LIN {X 0,Y 152.745,Z 601.305,A -85,B 0,C 180,E1 -23923.975,E2 -23923.975} C_VEL
LIN {X 0,Y 150.02,Z 597.18,A -85,B 0,C 180,E1 -23929.2,E2 -23929.2} C_VEL
LIN {X 0,Y 148.785,Z 591.816,A -85,B 0,C 180,E1 -23934.579,E2 -23934.579} C_VEL
LIN {X 0,Y 148.504,Z 586.8,A -85,B 0,C 180,E1 -23938.644,E2 -23938.644} C_VEL
LIN {X 0,Y 148.54,Z 579.677,A -85,B 0,C 180,E1 -23943.382,E2 -23943.382} C_VEL
LIN {X 0,Y 149.004,Z 570.731,A -85,B 0,C 180,E1 -23948.135,E2 -23948.135} C_VEL
LIN {X 0,Y 149.902,Z 561.531,A -85,B 0,C 180,E1 -23952.18,E2 -23952.18} C_VEL
LIN {X 0,Y 151.343,Z 550.54,A -85,B 0,C 180,E1 -23956.178,E2 -23956.178} C_VEL
LIN {X 0,Y 153.19,Z 538.222,A -85,B 0,C 180,E1 -23959.776,E2 -23959.776} C_VEL
LIN {X 0,Y 154.501,Z 528.967,A -85,B 0,C 180,E1 -23962.027,E2 -23962.027} C_VEL
LIN {X 0,Y 154.015,Z 524.912,A -85,B 0,C 180,E1 -23962.923,E2 -23962.923} C_VEL
LIN {X 0,Y 154.282,Z 525.794,A -85,B 0,C 180,E1 -23963.446,E2 -23963.446} C_VEL
LIN {X 0,Y 154.921,Z 526.142,A -85,B 0,C 180,E1 -23964.098,E2 -23964.098} C_VEL
LIN {X 0,Y 156.698,Z 525.145,A -85,B 0,C 180,E1 -23965.219,E2 -23965.219} C_VEL
LIN {X 0,Y 158.967,Z 522.474,A -85,B 0,C 180,E1 -23966.239,E2 -23966.239} C_VEL
LIN {X 0,Y 160.918,Z 521.843,A -85,B 0,C 180,E1 -23967.472,E2 -23967.472} C_VEL
LIN {X 0,Y 163.299,Z 519.845,A -85,B 0,C 180,E1 -23968.607,E2 -23968.607} C_VEL
LIN {X 0,Y 165.925,Z 516.496,A -85,B 0,C 180,E1 -23969.586,E2 -23969.586} C_VEL
LIN {X 0,Y 166.624,Z 515.781,A -85,B 0,C 180,E1 -23969.884,E2 -23969.884} C_VEL
LIN {X 0,Y 167.613,Z 515.285,A -85,B 0,C 180,E1 -23970.383,E2 -23970.383} C_VEL
LIN {X 0,Y 170.37,Z 518.349,A -85,B 0,C 180,E1 -23972.43,E2 -23972.43} C_VEL
LIN {X 0,Y 172.937,Z 522.605,A -85,B 0,C 180,E1 -23974.5,E2 -23974.5} C_VEL
LIN {X 0,Y 176.225,Z 530.359,A -85,B 0,C 180,E1 -23977.459,E2 -23977.459} C_VEL
LIN {X 0,Y 178.356,Z 536.742,A -85,B 0,C 180,E1 -23979.65,E2 -23979.65} C_VEL
LIN {X 0,Y 179.284,Z 542.682,A -85,B 0,C 180,E1 -23981.331,E2 -23981.331} C_VEL
LIN {X 0,Y 179.755,Z 554.232,A -85,B 0,C 180,E1 -23984.405,E2 -23984.405} C_VEL
LIN {X 0,Y 179.119,Z 565.311,A -85,B 0,C 180,E1 -23987.445,E2 -23987.445} C_VEL
LIN {X 0,Y 178.567,Z 569.644,A -85,B 0,C 180,E1 -23988.697,E2 -23988.697} C_VEL
LIN {X 0,Y 173.803,Z 580.088,A -85,B 0,C 180,E1 -23991.185,E2 -23991.185} C_VEL
LIN {X 0,Y 168.532,Z 590.306,A -85,B 0,C 180,E1 -23994.277,E2 -23994.277} C_VEL
LIN {X 0,Y 163.924,Z 598.73,A -85,B 0,C 180,E1 -23997.59,E2 -23997.59} C_VEL
LIN {X 0,Y 159.001,Z 606.865,A -85,B 0,C 180,E1 -24001.699,E2 -24001.699} C_VEL
LIN {X 0,Y 155.248,Z 613.225,A -85,B 0,C 180,E1 -24005.953,E2 -24005.953} C_VEL
LIN {X 0,Y 152.55,Z 617.694,A -85,B 0,C 180,E1 -24009.783,E2 -24009.783} C_VEL
LIN {X 0,Y 150.41,Z 621.2,A -85,B 0,C 180,E1 -24013.715,E2 -24013.715} C_VEL
LIN {X 0,Y 148.596,Z 624.62,A -85,B 0,C 180,E1 -24019.091,E2 -24019.091} C_VEL
LIN {X 0,Y 147.704,Z 626.652,A -85,B 0,C 180,E1 -24024.536,E2 -24024.536} C_VEL
LIN {X 0,Y 147.629,Z 627.344,A -85,B 0,C 180,E1 -24029.997,E2 -24029.997} C_VEL
LIN {X 0,Y 147.702,Z 626.705,A -85,B 0,C 180,E1 -24035.457,E2 -24035.457} C_VEL
LIN {X 0,Y 148.571,Z 624.718,A -85,B 0,C 180,E1 -24040.903,E2 -24040.903} C_VEL
LIN {X 0,Y 150.349,Z 621.341,A -85,B 0,C 180,E1 -24046.284,E2 -24046.284} C_VEL
LIN {X 0,Y 153.36,Z 616.469,A -85,B 0,C 180,E1 -24051.503,E2 -24051.503} C_VEL
LIN {X 0,Y 156.231,Z 611.748,A -85,B 0,C 180,E1 -24055.296,E2 -24055.296} C_VEL
LIN {X 0,Y 160.294,Z 604.906,A -85,B 0,C 180,E1 -24059.551,E2 -24059.551} C_VEL
LIN {X 0,Y 165.31,Z 596.406,A -85,B 0,C 180,E1 -24063.547,E2 -24063.547} C_VEL
LIN {X 0,Y 170.162,Z 587.512,A -85,B 0,C 180,E1 -24066.785,E2 -24066.785} C_VEL
LIN {X 0,Y 175.567,Z 576.736,A -85,B 0,C 180,E1 -24069.824,E2 -24069.824} C_VEL
LIN {X 0,Y 178.508,Z 570.135,A -85,B 0,C 180,E1 -24071.344,E2 -24071.344} C_VEL
LIN {X 0,Y 179.601,Z 561.031,A -85,B 0,C 180,E1 -24073.901,E2 -24073.901} C_VEL
LIN {X 0,Y 179.815,Z 552.025,A -85,B 0,C 180,E1 -24076.347,E2 -24076.347} C_VEL
LIN {X 0,Y 179.189,Z 541.022,A -85,B 0,C 180,E1 -24079.277,E2 -24079.277} C_VEL
LIN {X 0,Y 178.169,Z 535.607,A -85,B 0,C 180,E1 -24080.866,E2 -24080.866} C_VEL
LIN {X 0,Y 174.614,Z 526.074,A -85,B 0,C 180,E1 -24084.295,E2 -24084.295} C_VEL
LIN {X 0,Y 171.422,Z 519.258,A -85,B 0,C 180,E1 -24087.096,E2 -24087.096} C_VEL
LIN {X 0,Y 169.471,Z 515.528,A -85,B 0,C 180,E1 -24088.776,E2 -24088.776} C_VEL
LIN {X 0,Y 166.715,Z 510.789,A -85,B 0,C 180,E1 -24091.188,E2 -24091.188} C_VEL
LIN {X 0,Y 164.013,Z 506.647,A -85,B 0,C 180,E1 -24093.604,E2 -24093.604} C_VEL
LIN {X 0,Y 163.126,Z 505.162,A -85,B 0,C 180,E1 -24094.479,E2 -24094.479} C_VEL
LIN {X 0,Y 160.311,Z 501.441,A -85,B 0,C 180,E1 -24097.21,E2 -24097.21} C_VEL
LIN {X 0,Y 159.174,Z 499.399,A -85,B 0,C 180,E1 -24098.511,E2 -24098.511} C_VEL
LIN {X 0,Y 155.732,Z 495.52,A -85,B 0,C 180,E1 -24102.603,E2 -24102.603} C_VEL
LIN {X 0,Y 154.403,Z 493.061,A -85,B 0,C 180,E1 -24104.827,E2 -24104.827} C_VEL
LIN {X 0,Y 154.236,Z 491.472,A -85,B 0,C 180,E1 -24109.498,E2 -24109.498} C_VEL
LIN {X 0,Y 154.177,Z 490.844,A -85,B 0,C 180,E1 -24112.14,E2 -24112.14} C_VEL
LIN {X 0,Y 154.299,Z 489.663,A -85,B 0,C 180,E1 -24120,E2 -24120} C_VEL
LIN {X 0,Y 154.024,Z 490.167,A -85,B 0,C 180,E1 -24125.236,E2 -24125.236} C_VEL
LIN {X 0,Y 154.391,Z 491.072,A -85,B 0,C 180,E1 -24130.491,E2 -24130.491} C_VEL
LIN {X 0,Y 154.81,Z 492.811,A -85,B 0,C 180,E1 -24135.806,E2 -24135.806} C_VEL
LIN {X 0,Y 158.463,Z 497.876,A -85,B 0,C 180,E1 -24140.781,E2 -24140.781} C_VEL
LIN {X 0,Y 160.423,Z 499.793,A -85,B 0,C 180,E1 -24142.795,E2 -24142.795} C_VEL
LIN {X 0,Y 163.521,Z 504.046,A -85,B 0,C 180,E1 -24145.796,E2 -24145.796} C_VEL
LIN {X 0,Y 165.119,Z 505.889,A -85,B 0,C 180,E1 -24147.144,E2 -24147.144} C_VEL
LIN {X 0,Y 168.025,Z 510.29,A -85,B 0,C 180,E1 -24149.63,E2 -24149.63} C_VEL
LIN {X 0,Y 172.528,Z 517.457,A -85,B 0,C 180,E1 -24153.187,E2 -24153.187} C_VEL
LIN {X 0,Y 175.298,Z 522.617,A -85,B 0,C 180,E1 -24155.368,E2 -24155.368} C_VEL
LIN {X 0,Y 178.224,Z 530.027,A -85,B 0,C 180,E1 -24157.944,E2 -24157.944} C_VEL
LIN {X 0,Y 181.369,Z 540.405,A -85,B 0,C 180,E1 -24161.204,E2 -24161.204} C_VEL
LIN {X 0,Y 182.33,Z 544.543,A -85,B 0,C 180,E1 -24162.42,E2 -24162.42} C_VEL
LIN {X 0,Y 181.694,Z 553.891,A -85,B 0,C 180,E1 -24164.445,E2 -24164.445} C_VEL
LIN {X 0,Y 180.069,Z 564.713,A -85,B 0,C 180,E1 -24166.925,E2 -24166.925} C_VEL
LIN {X 0,Y 179.366,Z 568.481,A -85,B 0,C 180,E1 -24167.86,E2 -24167.86} C_VEL
LIN {X 0,Y 175.098,Z 578.414,A -85,B 0,C 180,E1 -24170.048,E2 -24170.048} C_VEL
LIN {X 0,Y 169.726,Z 589.325,A -85,B 0,C 180,E1 -24173.105,E2 -24173.105} C_VEL
LIN {X 0,Y 164.789,Z 598.321,A -85,B 0,C 180,E1 -24176.333,E2 -24176.333} C_VEL
LIN {X 0,Y 159.784,Z 606.913,A -85,B 0,C 180,E1 -24180.346,E2 -24180.346} C_VEL
LIN {X 0,Y 155.726,Z 613.69,A -85,B 0,C 180,E1 -24184.503,E2 -24184.503} C_VEL
LIN {X 0,Y 152.884,Z 618.613,A -85,B 0,C 180,E1 -24188.427,E2 -24188.427} C_VEL
LIN {X 0,Y 149.991,Z 623.544,A -85,B 0,C 180,E1 -24193.676,E2 -24193.676} C_VEL
LIN {X 0,Y 148.335,Z 626.972,A -85,B 0,C 180,E1 -24199.079,E2 -24199.079} C_VEL
LIN {X 0,Y 147.636,Z 628.996,A -85,B 0,C 180,E1 -24204.54,E2 -24204.54} C_VEL
LIN {X 0,Y 147.656,Z 629.662,A -85,B 0,C 180,E1 -24210.003,E2 -24210.003} C_VEL
LIN {X 0,Y 147.638,Z 628.969,A -85,B 0,C 180,E1 -24215.467,E2 -24215.467} C_VEL
LIN {X 0,Y 148.337,Z 626.921,A -85,B 0,C 180,E1 -24220.928,E2 -24220.928} C_VEL
LIN {X 0,Y 149.989,Z 623.472,A -85,B 0,C 180,E1 -24226.332,E2 -24226.332} C_VEL
LIN {X 0,Y 152.932,Z 618.521,A -85,B 0,C 180,E1 -24231.573,E2 -24231.573} C_VEL
LIN {X 0,Y 156.628,Z 612.797,A -85,B 0,C 180,E1 -24236.062,E2 -24236.062} C_VEL
LIN {X 0,Y 159.933,Z 612.793,A -85,B 0,C 180,E1 -24239.069,E2 -24239.069} C_VEL
LIN {X 0,Y 161.813,Z 612.596,A -85,B 0,C 180,E1 -24241.065,E2 -24241.065} C_VEL
LIN {X 0,Y 165.702,Z 611.319,A -85,B 0,C 180,E1 -24247.145,E2 -24247.145} C_VEL
LIN {X 0,Y 168.19,Z 610.693,A -85,B 0,C 180,E1 -24248.962,E2 -24248.962} C_VEL
LIN {X 0,Y 169.302,Z 610.438,A -85,B 0,C 180,E1 -24249.504,E2 -24249.504} C_VEL
LIN {X 0,Y 176.783,Z 608.741,A -85,B 0,C 180,E1 -24252.522,E2 -24252.522} C_VEL
LIN {X 0,Y 186.653,Z 605.968,A -85,B 0,C 180,E1 -24255.68,E2 -24255.68} C_VEL
LIN {X 0,Y 191.903,Z 604.248,A -85,B 0,C 180,E1 -24257.096,E2 -24257.096} C_VEL
LIN {X 0,Y 189.7,Z 604.678,A -85,B 0,C 180,E1 -24258.175,E2 -24258.175} C_VEL
LIN {X 0,Y 179.707,Z 606.525,A -85,B 0,C 180,E1 -24261.264,E2 -24261.264} C_VEL
LIN {X 0,Y 170.593,Z 607.407,A -85,B 0,C 180,E1 -24264.777,E2 -24264.777} C_VEL
LIN {X 0,Y 162.576,Z 607.267,A -85,B 0,C 180,E1 -24268.752,E2 -24268.752} C_VEL
LIN {X 0,Y 155.648,Z 606.102,A -85,B 0,C 180,E1 -24273.158,E2 -24273.158} C_VEL
LIN {X 0,Y 150.111,Z 603.906,A -85,B 0,C 180,E1 -24278.004,E2 -24278.004} C_VEL
LIN {X 0,Y 145.974,Z 600.632,A -85,B 0,C 180,E1 -24283.21,E2 -24283.21} C_VEL
LIN {X 0,Y 143.118,Z 596.212,A -85,B 0,C 180,E1 -24288.672,E2 -24288.672} C_VEL
LIN {X 0,Y 141.842,Z 590.519,A -85,B 0,C 180,E1 -24294.313,E2 -24294.313} C_VEL
LIN {X 0,Y 141.562,Z 585.228,A -85,B 0,C 180,E1 -24298.578,E2 -24298.578} C_VEL
LIN {X 0,Y 141.586,Z 577.702,A -85,B 0,C 180,E1 -24303.558,E2 -24303.558} C_VEL
LIN {X 0,Y 142.091,Z 568.752,A -85,B 0,C 180,E1 -24308.398,E2 -24308.398} C_VEL
LIN {X 0,Y 143.055,Z 558.741,A -85,B 0,C 180,E1 -24312.772,E2 -24312.772} C_VEL
LIN {X 0,Y 144.643,Z 547.183,A -85,B 0,C 180,E1 -24316.95,E2 -24316.95} C_VEL
LIN {X 0,Y 146.232,Z 536.905,A -85,B 0,C 180,E1 -24320.025,E2 -24320.025} C_VEL
LIN {X 0,Y 146.286,Z 537.527,A -85,B 0,C 180,E1 -24320.384,E2 -24320.384} C_VEL
LIN {X 0,Y 146.757,Z 537.877,A -85,B 0,C 180,E1 -24321.049,E2 -24321.049} C_VEL
LIN {X 0,Y 148.425,Z 536.943,A -85,B 0,C 180,E1 -24322.26,E2 -24322.26} C_VEL
LIN {X 0,Y 149.796,Z 535.685,A -85,B 0,C 180,E1 -24323.025,E2 -24323.025} C_VEL
LIN {X 0,Y 151.371,Z 533.937,A -85,B 0,C 180,E1 -24323.746,E2 -24323.746} C_VEL
LIN {X 0,Y 152.714,Z 532.816,A -85,B 0,C 180,E1 -24324.468,E2 -24324.468} C_VEL
LIN {X 0,Y 156.409,Z 530.942,A -85,B 0,C 180,E1 -24326.701,E2 -24326.701} C_VEL
LIN {X 0,Y 158.649,Z 528.916,A -85,B 0,C 180,E1 -24327.721,E2 -24327.721} C_VEL
LIN {X 0,Y 160.605,Z 527.941,A -85,B 0,C 180,E1 -24328.774,E2 -24328.774} C_VEL
LIN {X 0,Y 164.033,Z 525.175,A -85,B 0,C 180,E1 -24330.227,E2 -24330.227} C_VEL
LIN {X 0,Y 165.296,Z 523.852,A -85,B 0,C 180,E1 -24330.678,E2 -24330.678} C_VEL
LIN {X 0,Y 167.001,Z 524.279,A -85,B 0,C 180,E1 -24331.739,E2 -24331.739} C_VEL
LIN {X 0,Y 169.286,Z 528.465,A -85,B 0,C 180,E1 -24333.865,E2 -24333.865} C_VEL
LIN {X 0,Y 172.37,Z 536.848,A -85,B 0,C 180,E1 -24337.198,E2 -24337.198} C_VEL
LIN {X 0,Y 173.831,Z 542.617,A -85,B 0,C 180,E1 -24339.216,E2 -24339.216} C_VEL
LIN {X 0,Y 174.268,Z 553.874,A -85,B 0,C 180,E1 -24342.418,E2 -24342.418} C_VEL
LIN {X 0,Y 173.604,Z 564.648,A -85,B 0,C 180,E1 -24345.522,E2 -24345.522} C_VEL
LIN {X 0,Y 172.754,Z 570.8,A -85,B 0,C 180,E1 -24347.362,E2 -24347.362} C_VEL
LIN {X 0,Y 167.375,Z 581.991,A -85,B 0,C 180,E1 -24350.179,E2 -24350.179} C_VEL
LIN {X 0,Y 161.971,Z 591.842,A -85,B 0,C 180,E1 -24353.368,E2 -24353.368} C_VEL
LIN {X 0,Y 157.167,Z 600.013,A -85,B 0,C 180,E1 -24356.782,E2 -24356.782} C_VEL
LIN {X 0,Y 152.177,Z 607.817,A -85,B 0,C 180,E1 -24360.989,E2 -24360.989} C_VEL
LIN {X 0,Y 148.745,Z 613.281,A -85,B 0,C 180,E1 -24364.831,E2 -24364.831} C_VEL
LIN {X 0,Y 145.896,Z 617.75,A -85,B 0,C 180,E1 -24368.817,E2 -24368.817} C_VEL
LIN {X 0,Y 143.566,Z 621.257,A -85,B 0,C 180,E1 -24372.916,E2 -24372.916} C_VEL
LIN {X 0,Y 141.619,Z 624.676,A -85,B 0,C 180,E1 -24378.547,E2 -24378.547} C_VEL
LIN {X 0,Y 140.636,Z 626.708,A -85,B 0,C 180,E1 -24384.26,E2 -24384.26} C_VEL
LIN {X 0,Y 140.524,Z 627.4,A -85,B 0,C 180,E1 -24389.996,E2 -24389.996} C_VEL
LIN {X 0,Y 140.634,Z 626.76,A -85,B 0,C 180,E1 -24395.732,E2 -24395.732} C_VEL
LIN {X 0,Y 141.597,Z 624.773,A -85,B 0,C 180,E1 -24401.448,E2 -24401.448} C_VEL
LIN {X 0,Y 143.501,Z 621.396,A -85,B 0,C 180,E1 -24407.085,E2 -24407.085} C_VEL
LIN {X 0,Y 146.762,Z 616.522,A -85,B 0,C 180,E1 -24412.522,E2 -24412.522} C_VEL
LIN {X 0,Y 150.794,Z 610.123,A -85,B 0,C 180,E1 -24417.683,E2 -24417.683} C_VEL
LIN {X 0,Y 155.566,Z 602.746,A -85,B 0,C 180,E1 -24422.057,E2 -24422.057} C_VEL
LIN {X 0,Y 161.06,Z 593.681,A -85,B 0,C 180,E1 -24426.088,E2 -24426.088} C_VEL
LIN {X 0,Y 166.367,Z 584.194,A -85,B 0,C 180,E1 -24429.316,E2 -24429.316} C_VEL
LIN {X 0,Y 171.48,Z 574.058,A -85,B 0,C 180,E1 -24432.003,E2 -24432.003} C_VEL
LIN {X 0,Y 172.75,Z 571.285,A -85,B 0,C 180,E1 -24432.659,E2 -24432.659} C_VEL
LIN {X 0,Y 174.058,Z 561.239,A -85,B 0,C 180,E1 -24435.63,E2 -24435.63} C_VEL
LIN {X 0,Y 174.325,Z 550.149,A -85,B 0,C 180,E1 -24438.813,E2 -24438.813} C_VEL
LIN {X 0,Y 173.824,Z 541.825,A -85,B 0,C 180,E1 -24441.192,E2 -24441.192} C_VEL
LIN {X 0,Y 171.35,Z 533.555,A -85,B 0,C 180,E1 -24444.234,E2 -24444.234} C_VEL
LIN {X 0,Y 168.565,Z 526.48,A -85,B 0,C 180,E1 -24447.179,E2 -24447.179} C_VEL
LIN {X 0,Y 165.933,Z 520.951,A -85,B 0,C 180,E1 -24449.804,E2 -24449.804} C_VEL
LIN {X 0,Y 163.599,Z 516.61,A -85,B 0,C 180,E1 -24452.149,E2 -24452.149} C_VEL
LIN {X 0,Y 161.136,Z 512.254,A -85,B 0,C 180,E1 -24454.747,E2 -24454.747} C_VEL
LIN {X 0,Y 157.588,Z 506.669,A -85,B 0,C 180,E1 -24458.773,E2 -24458.773} C_VEL
LIN {X 0,Y 156.741,Z 505.475,A -85,B 0,C 180,E1 -24459.837,E2 -24459.837} C_VEL
LIN {X 0,Y 153.629,Z 501.238,A -85,B 0,C 180,E1 -24464.17,E2 -24464.17} C_VEL
LIN {X 0,Y 152.913,Z 499.845,A -85,B 0,C 180,E1 -24465.459,E2 -24465.459} C_VEL
LIN {X 0,Y 149.437,Z 496.006,A -85,B 0,C 180,E1 -24473.587,E2 -24473.587} C_VEL
LIN {X 0,Y 148.713,Z 494.072,A -85,B 0,C 180,E1 -24480,E2 -24480} C_VEL
LIN {X 0,Y 149.513,Z 495.771,A -85,B 0,C 180,E1 -24486.748,E2 -24486.748} C_VEL
LIN {X 0,Y 152.57,Z 498.99,A -85,B 0,C 180,E1 -24493.995,E2 -24493.995} C_VEL
LIN {X 0,Y 153.552,Z 499.951,A -85,B 0,C 180,E1 -24495.598,E2 -24495.598} C_VEL
LIN {X 0,Y 156.775,Z 504.534,A -85,B 0,C 180,E1 -24500.158,E2 -24500.158} C_VEL
LIN {X 0,Y 158.463,Z 506.364,A -85,B 0,C 180,E1 -24502.061,E2 -24502.061} C_VEL
LIN {X 0,Y 161.355,Z 510.575,A -85,B 0,C 180,E1 -24505.192,E2 -24505.192} C_VEL
LIN {X 0,Y 162.68,Z 512.363,A -85,B 0,C 180,E1 -24506.456,E2 -24506.456} C_VEL
LIN {X 0,Y 166.108,Z 518.009,A -85,B 0,C 180,E1 -24509.724,E2 -24509.724} C_VEL
LIN {X 0,Y 169.364,Z 523.761,A -85,B 0,C 180,E1 -24512.646,E2 -24512.646} C_VEL
LIN {X 0,Y 171.875,Z 528.916,A -85,B 0,C 180,E1 -24514.922,E2 -24514.922} C_VEL
LIN {X 0,Y 175.232,Z 539.75,A -85,B 0,C 180,E1 -24518.711,E2 -24518.711} C_VEL
LIN {X 0,Y 177.008,Z 547.706,A -85,B 0,C 180,E1 -24521.29,E2 -24521.29} C_VEL
LIN {X 0,Y 176.036,Z 557.292,A -85,B 0,C 180,E1 -24523.48,E2 -24523.48} C_VEL
LIN {X 0,Y 173.914,Z 568.438,A -85,B 0,C 180,E1 -24526.213,E2 -24526.213} C_VEL
LIN {X 0,Y 173.18,Z 570.691,A -85,B 0,C 180,E1 -24526.757,E2 -24526.757} C_VEL
LIN {X 0,Y 167.806,Z 582.247,A -85,B 0,C 180,E1 -24529.526,E2 -24529.526} C_VEL
LIN {X 0,Y 162.263,Z 592.5,A -85,B 0,C 180,E1 -24532.677,E2 -24532.677} C_VEL
LIN {X 0,Y 157.312,Z 600.952,A -85,B 0,C 180,E1 -24536.056,E2 -24536.056} C_VEL
LIN {X 0,Y 152.27,Z 609.008,A -85,B 0,C 180,E1 -24540.258,E2 -24540.258} C_VEL
LIN {X 0,Y 148.193,Z 615.486,A -85,B 0,C 180,E1 -24544.738,E2 -24544.738} C_VEL
LIN {X 0,Y 144.601,Z 621.221,A -85,B 0,C 180,E1 -24550.114,E2 -24550.114} C_VEL
LIN {X 0,Y 142.117,Z 625.384,A -85,B 0,C 180,E1 -24555.688,E2 -24555.688} C_VEL
LIN {X 0,Y 140.836,Z 628.1,A -85,B 0,C 180,E1 -24561.394,E2 -24561.394} C_VEL
LIN {X 0,Y 140.486,Z 629.443,A -85,B 0,C 180,E1 -24567.136,E2 -24567.136} C_VEL
LIN {X 0,Y 140.56,Z 629.606,A -85,B 0,C 180,E1 -24570.004,E2 -24570.004} C_VEL
LIN {X 0,Y 140.557,Z 628.913,A -85,B 0,C 180,E1 -24575.743,E2 -24575.743} C_VEL
LIN {X 0,Y 141.349,Z 626.865,A -85,B 0,C 180,E1 -24581.475,E2 -24581.475} C_VEL
LIN {X 0,Y 143.148,Z 623.416,A -85,B 0,C 180,E1 -24587.136,E2 -24587.136} C_VEL
LIN {X 0,Y 146.308,Z 618.466,A -85,B 0,C 180,E1 -24592.603,E2 -24592.603} C_VEL
LIN {X 0,Y 150.818,Z 612.04,A -85,B 0,C 180,E1 -24597.778,E2 -24597.778} C_VEL
LIN {X 0,Y 156.729,Z 612.125,A -85,B 0,C 180,E1 -24602.558,E2 -24602.558} C_VEL
LIN {X 0,Y 163.918,Z 611.406,A -85,B 0,C 180,E1 -24606.891,E2 -24606.891} C_VEL
LIN {X 0,Y 169.302,Z 610.438,A -85,B 0,C 180,E1 -24609.504,E2 -24609.504} C_VEL
LIN {X 0,Y 171.201,Z 609.973,A -85,B 0,C 180,E1 -24610.678,E2 -24610.678} C_VEL
LIN {X 0,Y 175.043,Z 608.476,A -85,B 0,C 180,E1 -24614.936,E2 -24614.936} C_VEL
LIN {X 0,Y 177.34,Z 607.83,A -85,B 0,C 180,E1 -24615.967,E2 -24615.967} C_VEL
LIN {X 0,Y 181.798,Z 606.719,A -85,B 0,C 180,E1 -24617.269,E2 -24617.269} C_VEL
LIN {X 0,Y 179.334,Z 607.072,A -85,B 0,C 180,E1 -24618.224,E2 -24618.224} C_VEL
LIN {X 0,Y 169.455,Z 607.978,A -85,B 0,C 180,E1 -24621.53,E2 -24621.53} C_VEL
LIN {X 0,Y 160.535,Z 607.925,A -85,B 0,C 180,E1 -24625.311,E2 -24625.311} C_VEL
LIN {X 0,Y 152.833,Z 606.875,A -85,B 0,C 180,E1 -24629.613,E2 -24629.613} C_VEL
LIN {X 0,Y 146.216,Z 604.832,A -85,B 0,C 180,E1 -24634.368,E2 -24634.368} C_VEL
LIN {X 0,Y 141.255,Z 601.773,A -85,B 0,C 180,E1 -24639.618,E2 -24639.618} C_VEL
LIN {X 0,Y 137.629,Z 597.602,A -85,B 0,C 180,E1 -24645.207,E2 -24645.207} C_VEL
LIN {X 0,Y 135.447,Z 592.235,A -85,B 0,C 180,E1 -24651.045,E2 -24651.045} C_VEL
LIN {X 0,Y 134.706,Z 585.453,A -85,B 0,C 180,E1 -24657.01,E2 -24657.01} C_VEL
LIN {X 0,Y 134.636,Z 579.214,A -85,B 0,C 180,E1 -24661.496,E2 -24661.496} C_VEL
LIN {X 0,Y 134.854,Z 571.668,A -85,B 0,C 180,E1 -24665.983,E2 -24665.983} C_VEL
LIN {X 0,Y 135.542,Z 562.732,A -85,B 0,C 180,E1 -24670.455,E2 -24670.455} C_VEL
LIN {X 0,Y 136.746,Z 552,A -85,B 0,C 180,E1 -24674.891,E2 -24674.891} C_VEL
LIN {X 0,Y 137.304,Z 548.57,A -85,B 0,C 180,E1 -24676.16,E2 -24676.16} C_VEL
LIN {X 0,Y 137.271,Z 548.882,A -85,B 0,C 180,E1 -24676.355,E2 -24676.355} C_VEL
LIN {X 0,Y 138.091,Z 549.29,A -85,B 0,C 180,E1 -24677.78,E2 -24677.78} C_VEL
LIN {X 0,Y 139.693,Z 548.271,A -85,B 0,C 180,E1 -24679.088,E2 -24679.088} C_VEL
LIN {X 0,Y 142.929,Z 545.227,A -85,B 0,C 180,E1 -24680.883,E2 -24680.883} C_VEL
LIN {X 0,Y 147.474,Z 542.551,A -85,B 0,C 180,E1 -24683.896,E2 -24683.896} C_VEL
LIN {X 0,Y 152.006,Z 538.7,A -85,B 0,C 180,E1 -24686.055,E2 -24686.055} C_VEL
LIN {X 0,Y 155.4,Z 537.086,A -85,B 0,C 180,E1 -24687.955,E2 -24687.955} C_VEL
LIN {X 0,Y 158.292,Z 534.927,A -85,B 0,C 180,E1 -24689.235,E2 -24689.235} C_VEL
LIN {X 0,Y 160.451,Z 533.712,A -85,B 0,C 180,E1 -24690.247,E2 -24690.247} C_VEL
LIN {X 0,Y 164.02,Z 531.183,A -85,B 0,C 180,E1 -24691.661,E2 -24691.661} C_VEL
LIN {X 0,Y 165.898,Z 535.484,A -85,B 0,C 180,E1 -24693.788,E2 -24693.788} C_VEL
LIN {X 0,Y 168.368,Z 543.984,A -85,B 0,C 180,E1 -24697.249,E2 -24697.249} C_VEL
LIN {X 0,Y 168.886,Z 548.053,A -85,B 0,C 180,E1 -24698.624,E2 -24698.624} C_VEL
LIN {X 0,Y 168.71,Z 558.573,A -85,B 0,C 180,E1 -24701.799,E2 -24701.799} C_VEL
LIN {X 0,Y 167.499,Z 569.259,A -85,B 0,C 180,E1 -24705.099,E2 -24705.099} C_VEL
LIN {X 0,Y 166.621,Z 573.022,A -85,B 0,C 180,E1 -24706.246,E2 -24706.246} C_VEL
LIN {X 0,Y 160.983,Z 583.799,A -85,B 0,C 180,E1 -24709.088,E2 -24709.088} C_VEL
LIN {X 0,Y 155.433,Z 593.361,A -85,B 0,C 180,E1 -24712.377,E2 -24712.377} C_VEL
LIN {X 0,Y 150.456,Z 601.283,A -85,B 0,C 180,E1 -24715.903,E2 -24715.903} C_VEL
LIN {X 0,Y 145.977,Z 607.872,A -85,B 0,C 180,E1 -24719.631,E2 -24719.631} C_VEL
LIN {X 0,Y 142.308,Z 613.336,A -85,B 0,C 180,E1 -24723.607,E2 -24723.607} C_VEL
LIN {X 0,Y 139.275,Z 617.806,A -85,B 0,C 180,E1 -24727.758,E2 -24727.758} C_VEL
LIN {X 0,Y 136.755,Z 621.313,A -85,B 0,C 180,E1 -24732.037,E2 -24732.037} C_VEL
LIN {X 0,Y 134.635,Z 624.733,A -85,B 0,C 180,E1 -24737.944,E2 -24737.944} C_VEL
LIN {X 0,Y 133.565,Z 626.764,A -85,B 0,C 180,E1 -24743.955,E2 -24743.955} C_VEL
LIN {X 0,Y 133.449,Z 627.456,A -85,B 0,C 180,E1 -24749.996,E2 -24749.996} C_VEL
LIN {X 0,Y 133.563,Z 626.816,A -85,B 0,C 180,E1 -24756.037,E2 -24756.037} C_VEL
LIN {X 0,Y 134.613,Z 624.828,A -85,B 0,C 180,E1 -24762.05,E2 -24762.05} C_VEL
LIN {X 0,Y 136.688,Z 621.45,A -85,B 0,C 180,E1 -24767.965,E2 -24767.965} C_VEL
LIN {X 0,Y 140.211,Z 616.576,A -85,B 0,C 180,E1 -24773.636,E2 -24773.636} C_VEL
LIN {X 0,Y 144.23,Z 610.573,A -85,B 0,C 180,E1 -24778.705,E2 -24778.705} C_VEL
LIN {X 0,Y 148.794,Z 603.906,A -85,B 0,C 180,E1 -24782.896,E2 -24782.896} C_VEL
LIN {X 0,Y 154.489,Z 595.167,A -85,B 0,C 180,E1 -24787.064,E2 -24787.064} C_VEL
LIN {X 0,Y 159.943,Z 585.99,A -85,B 0,C 180,E1 -24790.396,E2 -24790.396} C_VEL
LIN {X 0,Y 165.74,Z 575.184,A -85,B 0,C 180,E1 -24793.385,E2 -24793.385} C_VEL
LIN {X 0,Y 167.008,Z 572.408,A -85,B 0,C 180,E1 -24794.071,E2 -24794.071} C_VEL
LIN {X 0,Y 168.517,Z 562.658,A -85,B 0,C 180,E1 -24797.111,E2 -24797.111} C_VEL
LIN {X 0,Y 169.011,Z 552.414,A -85,B 0,C 180,E1 -24800.24,E2 -24800.24} C_VEL
LIN {X 0,Y 168.852,Z 545.761,A -85,B 0,C 180,E1 -24802.257,E2 -24802.257} C_VEL
LIN {X 0,Y 166.984,Z 538.487,A -85,B 0,C 180,E1 -24805.119,E2 -24805.119} C_VEL
LIN {X 0,Y 164.384,Z 531.084,A -85,B 0,C 180,E1 -24808.417,E2 -24808.417} C_VEL
LIN {X 0,Y 162.342,Z 526.409,A -85,B 0,C 180,E1 -24810.783,E2 -24810.783} C_VEL
LIN {X 0,Y 160.32,Z 522.349,A -85,B 0,C 180,E1 -24813.123,E2 -24813.123} C_VEL
LIN {X 0,Y 157.835,Z 517.532,A -85,B 0,C 180,E1 -24816.201,E2 -24816.201} C_VEL
LIN {X 0,Y 155.161,Z 512.725,A -85,B 0,C 180,E1 -24819.795,E2 -24819.795} C_VEL
LIN {X 0,Y 151.772,Z 507.582,A -85,B 0,C 180,E1 -24825.141,E2 -24825.141} C_VEL
LIN {X 0,Y 151.082,Z 506.372,A -85,B 0,C 180,E1 -24826.55,E2 -24826.55} C_VEL
LIN {X 0,Y 148.344,Z 502.979,A -85,B 0,C 180,E1 -24833.881,E2 -24833.881} C_VEL
LIN {X 0,Y 147.766,Z 501.132,A -85,B 0,C 180,E1 -24840,E2 -24840} C_VEL
LIN {X 0,Y 148.212,Z 502.45,A -85,B 0,C 180,E1 -24845.442,E2 -24845.442} C_VEL
LIN {X 0,Y 150.633,Z 505.263,A -85,B 0,C 180,E1 -24852.461,E2 -24852.461} C_VEL
LIN {X 0,Y 152.017,Z 506.815,A -85,B 0,C 180,E1 -24855.073,E2 -24855.073} C_VEL
LIN {X 0,Y 155.075,Z 511.457,A -85,B 0,C 180,E1 -24859.871,E2 -24859.871} C_VEL
LIN {X 0,Y 156.309,Z 512.995,A -85,B 0,C 180,E1 -24861.427,E2 -24861.427} C_VEL
LIN {X 0,Y 158.981,Z 517.094,A -85,B 0,C 180,E1 -24864.658,E2 -24864.658} C_VEL
LIN {X 0,Y 160.45,Z 519.696,A -85,B 0,C 180,E1 -24866.327,E2 -24866.327} C_VEL
LIN {X 0,Y 162.828,Z 523.823,A -85,B 0,C 180,E1 -24868.873,E2 -24868.873} C_VEL
LIN {X 0,Y 165.336,Z 528.599,A -85,B 0,C 180,E1 -24871.463,E2 -24871.463} C_VEL
LIN {X 0,Y 167.531,Z 533.495,A -85,B 0,C 180,E1 -24873.769,E2 -24873.769} C_VEL
LIN {X 0,Y 169.841,Z 541.645,A -85,B 0,C 180,E1 -24876.87,E2 -24876.87} C_VEL
LIN {X 0,Y 171.587,Z 549.961,A -85,B 0,C 180,E1 -24879.789,E2 -24879.789} C_VEL
LIN {X 0,Y 171.56,Z 552.804,A -85,B 0,C 180,E1 -24880.587,E2 -24880.587} C_VEL
LIN {X 0,Y 169.767,Z 563.352,A -85,B 0,C 180,E1 -24883.149,E2 -24883.149} C_VEL
LIN {X 0,Y 167.968,Z 570.865,A -85,B 0,C 180,E1 -24885.139,E2 -24885.139} C_VEL
LIN {X 0,Y 162.45,Z 582.202,A -85,B 0,C 180,E1 -24887.894,E2 -24887.894} C_VEL
LIN {X 0,Y 156.675,Z 592.452,A -85,B 0,C 180,E1 -24891.102,E2 -24891.102} C_VEL
LIN {X 0,Y 151.449,Z 600.902,A -85,B 0,C 180,E1 -24894.55,E2 -24894.55} C_VEL
LIN {X 0,Y 146.115,Z 608.956,A -85,B 0,C 180,E1 -24898.869,E2 -24898.869} C_VEL
LIN {X 0,Y 141.74,Z 615.433,A -85,B 0,C 180,E1 -24903.501,E2 -24903.501} C_VEL
LIN {X 0,Y 137.91,Z 621.167,A -85,B 0,C 180,E1 -24909.105,E2 -24909.105} C_VEL
LIN {X 0,Y 135.205,Z 625.329,A -85,B 0,C 180,E1 -24914.94,E2 -24914.94} C_VEL
LIN {X 0,Y 133.808,Z 628.044,A -85,B 0,C 180,E1 -24920.938,E2 -24920.938} C_VEL
LIN {X 0,Y 133.397,Z 629.387,A -85,B 0,C 180,E1 -24926.984,E2 -24926.984} C_VEL
LIN {X 0,Y 133.456,Z 629.55,A -85,B 0,C 180,E1 -24930.004,E2 -24930.004} C_VEL
LIN {X 0,Y 133.398,Z 629.373,A -85,B 0,C 180,E1 -24933.024,E2 -24933.024} C_VEL
LIN {X 0,Y 133.81,Z 628.003,A -85,B 0,C 180,E1 -24939.069,E2 -24939.069} C_VEL
LIN {X 0,Y 135.206,Z 625.264,A -85,B 0,C 180,E1 -24945.068,E2 -24945.068} C_VEL
LIN {X 0,Y 137.924,Z 621.081,A -85,B 0,C 180,E1 -24950.901,E2 -24950.901} C_VEL
LIN {X 0,Y 141.966,Z 615.325,A -85,B 0,C 180,E1 -24956.462,E2 -24956.462} C_VEL
LIN {X 0,Y 145.134,Z 611.204,A -85,B 0,C 180,E1 -24959.563,E2 -24959.563} C_VEL
LIN {X 0,Y 154.396,Z 611.436,A -85,B 0,C 180,E1 -24966.285,E2 -24966.285} C_VEL
LIN {X 0,Y 163.749,Z 610.478,A -85,B 0,C 180,E1 -24971.014,E2 -24971.014} C_VEL
LIN {X 0,Y 171.624,Z 609.1,A -85,B 0,C 180,E1 -24974.122,E2 -24974.122} C_VEL
LIN {X 0,Y 177.34,Z 607.83,A -85,B 0,C 180,E1 -24975.967,E2 -24975.967} C_VEL
LIN {X 0,Y 177.752,Z 607.692,A -85,B 0,C 180,E1 -24976.381,E2 -24976.381} C_VEL
LIN {X 0,Y 176.861,Z 607.685,A -85,B 0,C 180,E1 -24977.142,E2 -24977.142} C_VEL
LIN {X 0,Y 174.26,Z 607.966,A -85,B 0,C 180,E1 -24978.01,E2 -24978.01} C_VEL
LIN {X 0,Y 163.604,Z 608.683,A -85,B 0,C 180,E1 -24980.236,E2 -24980.236} C_VEL
LIN {X 0,Y 161.718,Z 608.638,A -85,B 0,C 180,E1 -24980.859,E2 -24980.859} C_VEL
LIN {X 0,Y 154.772,Z 608.225,A -85,B 0,C 180,E1 -24983.821,E2 -24983.821} C_VEL
LIN {X 0,Y 146.772,Z 606.802,A -85,B 0,C 180,E1 -24988.216,E2 -24988.216} C_VEL
LIN {X 0,Y 139.871,Z 604.391,A -85,B 0,C 180,E1 -24993.114,E2 -24993.114} C_VEL
LIN {X 0,Y 134.662,Z 600.992,A -85,B 0,C 180,E1 -24998.572,E2 -24998.572} C_VEL
LIN {X 0,Y 130.874,Z 596.515,A -85,B 0,C 180,E1 -25004.425,E2 -25004.425} C_VEL
LIN {X 0,Y 128.597,Z 590.776,A -85,B 0,C 180,E1 -25010.564,E2 -25010.564} C_VEL
LIN {X 0,Y 127.93,Z 585.599,A -85,B 0,C 180,E1 -25015.273,E2 -25015.273} C_VEL
LIN {X 0,Y 127.727,Z 578.275,A -85,B 0,C 180,E1 -25020.788,E2 -25020.788} C_VEL
LIN {X 0,Y 127.904,Z 570.665,A -85,B 0,C 180,E1 -25025.518,E2 -25025.518} C_VEL
LIN {X 0,Y 128.588,Z 561.333,A -85,B 0,C 180,E1 -25030.311,E2 -25030.311} C_VEL
LIN {X 0,Y 128.872,Z 558.449,A -85,B 0,C 180,E1 -25031.7,E2 -25031.7} C_VEL
LIN {X 0,Y 128.934,Z 559.016,A -85,B 0,C 180,E1 -25032.594,E2 -25032.594} C_VEL
LIN {X 0,Y 131.365,Z 557.779,A -85,B 0,C 180,E1 -25035.516,E2 -25035.516} C_VEL
LIN {X 0,Y 133.313,Z 556.147,A -85,B 0,C 180,E1 -25036.855,E2 -25036.855} C_VEL
LIN {X 0,Y 138.082,Z 553.645,A -85,B 0,C 180,E1 -25040.872,E2 -25040.872} C_VEL
LIN {X 0,Y 140.843,Z 551.371,A -85,B 0,C 180,E1 -25042.32,E2 -25042.32} C_VEL
LIN {X 0,Y 146.438,Z 548.042,A -85,B 0,C 180,E1 -25045.591,E2 -25045.591} C_VEL
LIN {X 0,Y 151.2,Z 544.457,A -85,B 0,C 180,E1 -25047.699,E2 -25047.699} C_VEL
LIN {X 0,Y 153.254,Z 543.563,A -85,B 0,C 180,E1 -25048.785,E2 -25048.785} C_VEL
LIN {X 0,Y 160.201,Z 539.388,A -85,B 0,C 180,E1 -25051.766,E2 -25051.766} C_VEL
LIN {X 0,Y 161.619,Z 540.577,A -85,B 0,C 180,E1 -25052.927,E2 -25052.927} C_VEL
LIN {X 0,Y 163.507,Z 548.197,A -85,B 0,C 180,E1 -25056.229,E2 -25056.229} C_VEL
LIN {X 0,Y 163.741,Z 552.719,A -85,B 0,C 180,E1 -25057.809,E2 -25057.809} C_VEL
LIN {X 0,Y 163.131,Z 562.228,A -85,B 0,C 180,E1 -25060.856,E2 -25060.856} C_VEL
LIN {X 0,Y 161.576,Z 572.122,A -85,B 0,C 180,E1 -25064.103,E2 -25064.103} C_VEL
LIN {X 0,Y 160.996,Z 574.174,A -85,B 0,C 180,E1 -25064.764,E2 -25064.764} C_VEL
LIN {X 0,Y 155.675,Z 583.851,A -85,B 0,C 180,E1 -25067.373,E2 -25067.373} C_VEL
LIN {X 0,Y 150.751,Z 591.948,A -85,B 0,C 180,E1 -25070.128,E2 -25070.128} C_VEL
LIN {X 0,Y 144.604,Z 601.338,A -85,B 0,C 180,E1 -25074.319,E2 -25074.319} C_VEL
LIN {X 0,Y 139.87,Z 607.927,A -85,B 0,C 180,E1 -25078.153,E2 -25078.153} C_VEL
LIN {X 0,Y 135.952,Z 613.392,A -85,B 0,C 180,E1 -25082.269,E2 -25082.269} C_VEL
LIN {X 0,Y 132.699,Z 617.862,A -85,B 0,C 180,E1 -25086.592,E2 -25086.592} C_VEL
LIN {X 0,Y 129.983,Z 621.369,A -85,B 0,C 180,E1 -25091.066,E2 -25091.066} C_VEL
LIN {X 0,Y 127.676,Z 624.789,A -85,B 0,C 180,E1 -25097.276,E2 -25097.276} C_VEL
LIN {X 0,Y 126.49,Z 626.82,A -85,B 0,C 180,E1 -25103.616,E2 -25103.616} C_VEL
LIN {X 0,Y 126.36,Z 627.511,A -85,B 0,C 180,E1 -25109.996,E2 -25109.996} C_VEL
LIN {X 0,Y 126.487,Z 626.871,A -85,B 0,C 180,E1 -25116.376,E2 -25116.376} C_VEL
LIN {X 0,Y 127.655,Z 624.883,A -85,B 0,C 180,E1 -25122.718,E2 -25122.718} C_VEL
LIN {X 0,Y 129.917,Z 621.505,A -85,B 0,C 180,E1 -25128.936,E2 -25128.936} C_VEL
LIN {X 0,Y 133.695,Z 616.63,A -85,B 0,C 180,E1 -25134.864,E2 -25134.864} C_VEL
LIN {X 0,Y 137.758,Z 610.981,A -85,B 0,C 180,E1 -25139.855,E2 -25139.855} C_VEL
LIN {X 0,Y 142.872,Z 603.957,A -85,B 0,C 180,E1 -25144.446,E2 -25144.446} C_VEL
LIN {X 0,Y 148.872,Z 595.216,A -85,B 0,C 180,E1 -25148.715,E2 -25148.715} C_VEL
LIN {X 0,Y 154.606,Z 586.037,A -85,B 0,C 180,E1 -25152.101,E2 -25152.101} C_VEL
LIN {X 0,Y 160.346,Z 575.797,A -85,B 0,C 180,E1 -25154.995,E2 -25154.995} C_VEL
LIN {X 0,Y 161.36,Z 573.539,A -85,B 0,C 180,E1 -25155.583,E2 -25155.583} C_VEL
LIN {X 0,Y 163.042,Z 564.124,A -85,B 0,C 180,E1 -25158.697,E2 -25158.697} C_VEL
LIN {X 0,Y 163.855,Z 553.586,A -85,B 0,C 180,E1 -25162.092,E2 -25162.092} C_VEL
LIN {X 0,Y 163.896,Z 550.428,A -85,B 0,C 180,E1 -25163.106,E2 -25163.106} C_VEL
LIN {X 0,Y 163.091,Z 545.802,A -85,B 0,C 180,E1 -25164.955,E2 -25164.955} C_VEL
LIN {X 0,Y 160.976,Z 538.233,A -85,B 0,C 180,E1 -25168.405,E2 -25168.405} C_VEL
LIN {X 0,Y 158.717,Z 532.014,A -85,B 0,C 180,E1 -25171.647,E2 -25171.647} C_VEL
LIN {X 0,Y 157.419,Z 528.808,A -85,B 0,C 180,E1 -25173.483,E2 -25173.483} C_VEL
LIN {X 0,Y 154.13,Z 522.412,A -85,B 0,C 180,E1 -25178.078,E2 -25178.078} C_VEL
LIN {X 0,Y 152.316,Z 518.498,A -85,B 0,C 180,E1 -25181.156,E2 -25181.156} C_VEL
LIN {X 0,Y 149.775,Z 514.078,A -85,B 0,C 180,E1 -25185.911,E2 -25185.911} C_VEL
LIN {X 0,Y 149.14,Z 512.931,A -85,B 0,C 180,E1 -25187.411,E2 -25187.411} C_VEL
LIN {X 0,Y 146.906,Z 509.779,A -85,B 0,C 180,E1 -25194.509,E2 -25194.509} C_VEL
LIN {X 0,Y 146.553,Z 508.133,A -85,B 0,C 180,E1 -25200,E2 -25200} C_VEL
LIN {X 0,Y 146.945,Z 509.479,A -85,B 0,C 180,E1 -25205.489,E2 -25205.489} C_VEL
LIN {X 0,Y 149.097,Z 512.197,A -85,B 0,C 180,E1 -25212.246,E2 -25212.246} C_VEL
LIN {X 0,Y 150.127,Z 513.407,A -85,B 0,C 180,E1 -25214.4,E2 -25214.4} C_VEL
LIN {X 0,Y 152.848,Z 518.02,A -85,B 0,C 180,E1 -25219.298,E2 -25219.298} C_VEL
LIN {X 0,Y 153.902,Z 519.521,A -85,B 0,C 180,E1 -25220.814,E2 -25220.814} C_VEL
LIN {X 0,Y 156.814,Z 524.442,A -85,B 0,C 180,E1 -25224.756,E2 -25224.756} C_VEL
LIN {X 0,Y 160.611,Z 532.099,A -85,B 0,C 180,E1 -25229.49,E2 -25229.49} C_VEL
LIN {X 0,Y 163.262,Z 538.294,A -85,B 0,C 180,E1 -25232.724,E2 -25232.724} C_VEL
LIN {X 0,Y 165.446,Z 547.613,A -85,B 0,C 180,E1 -25236.492,E2 -25236.492} C_VEL
LIN {X 0,Y 166.426,Z 553.934,A -85,B 0,C 180,E1 -25238.84,E2 -25238.84} C_VEL
LIN {X 0,Y 164.743,Z 563.311,A -85,B 0,C 180,E1 -25241.251,E2 -25241.251} C_VEL
LIN {X 0,Y 162.512,Z 571.785,A -85,B 0,C 180,E1 -25243.565,E2 -25243.565} C_VEL
LIN {X 0,Y 157.234,Z 582.156,A -85,B 0,C 180,E1 -25246.152,E2 -25246.152} C_VEL
LIN {X 0,Y 151.203,Z 592.404,A -85,B 0,C 180,E1 -25249.408,E2 -25249.408} C_VEL
LIN {X 0,Y 145.705,Z 600.852,A -85,B 0,C 180,E1 -25252.925,E2 -25252.925} C_VEL
LIN {X 0,Y 140.051,Z 608.904,A -85,B 0,C 180,E1 -25257.358,E2 -25257.358} C_VEL
LIN {X 0,Y 135.343,Z 615.379,A -85,B 0,C 180,E1 -25262.142,E2 -25262.142} C_VEL
LIN {X 0,Y 131.27,Z 621.113,A -85,B 0,C 180,E1 -25267.994,E2 -25267.994} C_VEL
LIN {X 0,Y 128.327,Z 625.274,A -85,B 0,C 180,E1 -25274.112,E2 -25274.112} C_VEL
LIN {X 0,Y 126.772,Z 627.989,A -85,B 0,C 180,E1 -25280.431,E2 -25280.431} C_VEL
LIN {X 0,Y 126.302,Z 629.332,A -85,B 0,C 180,E1 -25286.814,E2 -25286.814} C_VEL
LIN {X 0,Y 126.362,Z 629.495,A -85,B 0,C 180,E1 -25290.004,E2 -25290.004} C_VEL
LIN {X 0,Y 126.303,Z 629.317,A -85,B 0,C 180,E1 -25293.194,E2 -25293.194} C_VEL
LIN {X 0,Y 126.775,Z 627.947,A -85,B 0,C 180,E1 -25299.577,E2 -25299.577} C_VEL
LIN {X 0,Y 128.328,Z 625.208,A -85,B 0,C 180,E1 -25305.896,E2 -25305.896} C_VEL
LIN {X 0,Y 131.289,Z 621.025,A -85,B 0,C 180,E1 -25312.011,E2 -25312.011} C_VEL
LIN {X 0,Y 135.619,Z 615.269,A -85,B 0,C 180,E1 -25317.805,E2 -25317.805} C_VEL
LIN {X 0,Y 139.806,Z 610.272,A -85,B 0,C 180,E1 -25321.651,E2 -25321.651} C_VEL
LIN {X 0,Y 148.745,Z 610.858,A -85,B 0,C 180,E1 -25327.9,E2 -25327.9} C_VEL
LIN {X 0,Y 157.147,Z 610.44,A -85,B 0,C 180,E1 -25332.136,E2 -25332.136} C_VEL
LIN {X 0,Y 169.022,Z 608.876,A -85,B 0,C 180,E1 -25336.595,E2 -25336.595} C_VEL
LIN {X 0,Y 170.294,Z 608.648,A -85,B 0,C 180,E1 -25336.994,E2 -25336.994} C_VEL
LIN {X 0,Y 170.987,Z 608.449,A -85,B 0,C 180,E1 -25337.633,E2 -25337.633} C_VEL
LIN {X 0,Y 161.718,Z 608.638,A -85,B 0,C 180,E1 -25340.859,E2 -25340.859} C_VEL
LIN {X 0,Y 157.362,Z 608.551,A -85,B 0,C 180,E1 -25342.29,E2 -25342.29} C_VEL
LIN {X 0,Y 149.245,Z 607.898,A -85,B 0,C 180,E1 -25344.399,E2 -25344.399} C_VEL
LIN {X 0,Y 141.506,Z 606.638,A -85,B 0,C 180,E1 -25346.768,E2 -25346.768} C_VEL
LIN {X 0,Y 137.839,Z 605.581,A -85,B 0,C 180,E1 -25348.613,E2 -25348.613} C_VEL
LIN {X 0,Y 133.604,Z 603.785,A -85,B 0,C 180,E1 -25351.743,E2 -25351.743} C_VEL
LIN {X 0,Y 127.001,Z 598.924,A -85,B 0,C 180,E1 -25358.919,E2 -25358.919} C_VEL
LIN {X 0,Y 123.376,Z 593.807,A -85,B 0,C 180,E1 -25365.147,E2 -25365.147} C_VEL
LIN {X 0,Y 121.473,Z 587.409,A -85,B 0,C 180,E1 -25371.684,E2 -25371.684} C_VEL
LIN {X 0,Y 120.922,Z 580.614,A -85,B 0,C 180,E1 -25377.502,E2 -25377.502} C_VEL
LIN {X 0,Y 120.874,Z 573.481,A -85,B 0,C 180,E1 -25382.5,E2 -25382.5} C_VEL
LIN {X 0,Y 121.082,Z 567.205,A -85,B 0,C 180,E1 -25386.353,E2 -25386.353} C_VEL
LIN {X 0,Y 120.991,Z 567.42,A -85,B 0,C 180,E1 -25386.672,E2 -25386.672} C_VEL
LIN {X 0,Y 122.227,Z 567.078,A -85,B 0,C 180,E1 -25389.933,E2 -25389.933} C_VEL
LIN {X 0,Y 125.1,Z 564.899,A -85,B 0,C 180,E1 -25392.987,E2 -25392.987} C_VEL
LIN {X 0,Y 128.228,Z 563.558,A -85,B 0,C 180,E1 -25396.755,E2 -25396.755} C_VEL
LIN {X 0,Y 131.092,Z 561.583,A -85,B 0,C 180,E1 -25398.764,E2 -25398.764} C_VEL
LIN {X 0,Y 134.488,Z 559.943,A -85,B 0,C 180,E1 -25401.457,E2 -25401.457} C_VEL
LIN {X 0,Y 136.649,Z 558.707,A -85,B 0,C 180,E1 -25402.849,E2 -25402.849} C_VEL
LIN {X 0,Y 138.817,Z 557.097,A -85,B 0,C 180,E1 -25403.893,E2 -25403.893} C_VEL
LIN {X 0,Y 145.335,Z 553.411,A -85,B 0,C 180,E1 -25407.348,E2 -25407.348} C_VEL
LIN {X 0,Y 150.302,Z 550.103,A -85,B 0,C 180,E1 -25409.405,E2 -25409.405} C_VEL
LIN {X 0,Y 154.948,Z 547.692,A -85,B 0,C 180,E1 -25411.44,E2 -25411.44} C_VEL
LIN {X 0,Y 157.391,Z 546.315,A -85,B 0,C 180,E1 -25412.401,E2 -25412.401} C_VEL
LIN {X 0,Y 158.57,Z 552.355,A -85,B 0,C 180,E1 -25415.182,E2 -25415.182} C_VEL
LIN {X 0,Y 158.614,Z 555.83,A -85,B 0,C 180,E1 -25416.463,E2 -25416.463} C_VEL
LIN {X 0,Y 157.423,Z 566.5,A -85,B 0,C 180,E1 -25420.098,E2 -25420.098} C_VEL
LIN {X 0,Y 155.79,Z 574.373,A -85,B 0,C 180,E1 -25422.865,E2 -25422.865} C_VEL
LIN {X 0,Y 154.891,Z 576.437,A -85,B 0,C 180,E1 -25423.445,E2 -25423.445} C_VEL
LIN {X 0,Y 148.392,Z 587.309,A -85,B 0,C 180,E1 -25426.624,E2 -25426.624} C_VEL
LIN {X 0,Y 142.507,Z 596.277,A -85,B 0,C 180,E1 -25430.121,E2 -25430.121} C_VEL
LIN {X 0,Y 136.284,Z 604.839,A -85,B 0,C 180,E1 -25434.535,E2 -25434.535} C_VEL
LIN {X 0,Y 130.744,Z 612.003,A -85,B 0,C 180,E1 -25439.551,E2 -25439.551} C_VEL
LIN {X 0,Y 126.189,Z 617.918,A -85,B 0,C 180,E1 -25445.306,E2 -25445.306} C_VEL
LIN {X 0,Y 123.258,Z 621.425,A -85,B 0,C 180,E1 -25449.99,E2 -25449.99} C_VEL
LIN {X 0,Y 120.745,Z 624.845,A -85,B 0,C 180,E1 -25456.533,E2 -25456.533} C_VEL
LIN {X 0,Y 119.439,Z 626.876,A -85,B 0,C 180,E1 -25463.237,E2 -25463.237} C_VEL
LIN {X 0,Y 119.279,Z 627.567,A -85,B 0,C 180,E1 -25469.996,E2 -25469.996} C_VEL
LIN {X 0,Y 119.436,Z 626.926,A -85,B 0,C 180,E1 -25476.754,E2 -25476.754} C_VEL
LIN {X 0,Y 120.725,Z 624.938,A -85,B 0,C 180,E1 -25483.461,E2 -25483.461} C_VEL
LIN {X 0,Y 123.187,Z 621.559,A -85,B 0,C 180,E1 -25490.013,E2 -25490.013} C_VEL
LIN {X 0,Y 127.236,Z 616.683,A -85,B 0,C 180,E1 -25496.22,E2 -25496.22} C_VEL
LIN {X 0,Y 132.309,Z 610.171,A -85,B 0,C 180,E1 -25502.08,E2 -25502.08} C_VEL
LIN {X 0,Y 137.921,Z 602.899,A -85,B 0,C 180,E1 -25506.775,E2 -25506.775} C_VEL
LIN {X 0,Y 144.323,Z 593.827,A -85,B 0,C 180,E1 -25511.097,E2 -25511.097} C_VEL
LIN {X 0,Y 150.48,Z 584.332,A -85,B 0,C 180,E1 -25514.467,E2 -25514.467} C_VEL
LIN {X 0,Y 155.77,Z 574.871,A -85,B 0,C 180,E1 -25517.139,E2 -25517.139} C_VEL
LIN {X 0,Y 157.72,Z 565.607,A -85,B 0,C 180,E1 -25520.375,E2 -25520.375} C_VEL
LIN {X 0,Y 158.765,Z 555.455,A -85,B 0,C 180,E1 -25523.852,E2 -25523.852} C_VEL
LIN {X 0,Y 158.736,Z 552.703,A -85,B 0,C 180,E1 -25524.86,E2 -25524.86} C_VEL
LIN {X 0,Y 157.399,Z 545.844,A -85,B 0,C 180,E1 -25528.028,E2 -25528.028} C_VEL
LIN {X 0,Y 155.448,Z 538.934,A -85,B 0,C 180,E1 -25531.659,E2 -25531.659} C_VEL
LIN {X 0,Y 153.886,Z 534.619,A -85,B 0,C 180,E1 -25534.286,E2 -25534.286} C_VEL
LIN {X 0,Y 151.559,Z 529.166,A -85,B 0,C 180,E1 -25538.224,E2 -25538.224} C_VEL
LIN {X 0,Y 149.494,Z 524.556,A -85,B 0,C 180,E1 -25542.207,E2 -25542.207} C_VEL
LIN {X 0,Y 147.221,Z 519.746,A -85,B 0,C 180,E1 -25547.595,E2 -25547.595} C_VEL
LIN {X 0,Y 145.223,Z 516.638,A -85,B 0,C 180,E1 -25554.794,E2 -25554.794} C_VEL
LIN {X 0,Y 145.002,Z 515.098,A -85,B 0,C 180,E1 -25560,E2 -25560} C_VEL
LIN {X 0,Y 145.476,Z 516.639,A -85,B 0,C 180,E1 -25566.24,E2 -25566.24} C_VEL
LIN {X 0,Y 147.903,Z 519.798,A -85,B 0,C 180,E1 -25573.569,E2 -25573.569} C_VEL
LIN {X 0,Y 150.463,Z 524.626,A -85,B 0,C 180,E1 -25578.908,E2 -25578.908} C_VEL
LIN {X 0,Y 153.452,Z 529.94,A -85,B 0,C 180,E1 -25583.663,E2 -25583.663} C_VEL
LIN {X 0,Y 156.894,Z 537.798,A -85,B 0,C 180,E1 -25588.759,E2 -25588.759} C_VEL
LIN {X 0,Y 159.073,Z 543.798,A -85,B 0,C 180,E1 -25592.017,E2 -25592.017} C_VEL
LIN {X 0,Y 160.566,Z 551.897,A -85,B 0,C 180,E1 -25595.482,E2 -25595.482} C_VEL
LIN {X 0,Y 161.15,Z 557.35,A -85,B 0,C 180,E1 -25597.63,E2 -25597.63} C_VEL
LIN {X 0,Y 158.806,Z 567.315,A -85,B 0,C 180,E1 -25600.321,E2 -25600.321} C_VEL
LIN {X 0,Y 156.98,Z 573.201,A -85,B 0,C 180,E1 -25602.016,E2 -25602.016} C_VEL
LIN {X 0,Y 151.125,Z 583.958,A -85,B 0,C 180,E1 -25604.836,E2 -25604.836} C_VEL
LIN {X 0,Y 144.844,Z 593.838,A -85,B 0,C 180,E1 -25608.157,E2 -25608.157} C_VEL
LIN {X 0,Y 139.164,Z 602.03,A -85,B 0,C 180,E1 -25611.788,E2 -25611.788} C_VEL
LIN {X 0,Y 133.314,Z 609.854,A -85,B 0,C 180,E1 -25616.395,E2 -25616.395} C_VEL
LIN {X 0,Y 129.047,Z 615.326,A -85,B 0,C 180,E1 -25620.655,E2 -25620.655} C_VEL
LIN {X 0,Y 124.683,Z 621.058,A -85,B 0,C 180,E1 -25626.766,E2 -25626.766} C_VEL
LIN {X 0,Y 121.461,Z 625.219,A -85,B 0,C 180,E1 -25633.188,E2 -25633.188} C_VEL
LIN {X 0,Y 119.738,Z 627.934,A -85,B 0,C 180,E1 -25639.863,E2 -25639.863} C_VEL
LIN {X 0,Y 119.198,Z 629.276,A -85,B 0,C 180,E1 -25646.624,E2 -25646.624} C_VEL
LIN {X 0,Y 119.279,Z 629.439,A -85,B 0,C 180,E1 -25650.004,E2 -25650.004} C_VEL
LIN {X 0,Y 119.332,Z 628.745,A -85,B 0,C 180,E1 -25656.769,E2 -25656.769} C_VEL
LIN {X 0,Y 120.45,Z 626.696,A -85,B 0,C 180,E1 -25663.501,E2 -25663.501} C_VEL
LIN {X 0,Y 122.861,Z 623.247,A -85,B 0,C 180,E1 -25670.077,E2 -25670.077} C_VEL
LIN {X 0,Y 126.822,Z 618.298,A -85,B 0,C 180,E1 -25676.321,E2 -25676.321} C_VEL
LIN {X 0,Y 130.69,Z 613.585,A -85,B 0,C 180,E1 -25680.637,E2 -25680.637} C_VEL
LIN {X 0,Y 134.487,Z 609.242,A -85,B 0,C 180,E1 -25683.731,E2 -25683.731} C_VEL
LIN {X 0,Y 143.226,Z 610.117,A -85,B 0,C 180,E1 -25689.639,E2 -25689.639} C_VEL
LIN {X 0,Y 151.981,Z 610.041,A -85,B 0,C 180,E1 -25693.923,E2 -25693.923} C_VEL
LIN {X 0,Y 160.026,Z 609.452,A -85,B 0,C 180,E1 -25697.025,E2 -25697.025} C_VEL
LIN {X 0,Y 159.968,Z 609.291,A -85,B 0,C 180,E1 -25697.888,E2 -25697.888} C_VEL
LIN {X 0,Y 149.106,Z 608.366,A -85,B 0,C 180,E1 -25702.212,E2 -25702.212} C_VEL
LIN {X 0,Y 140.812,Z 606.564,A -85,B 0,C 180,E1 -25706.701,E2 -25706.701} C_VEL
LIN {X 0,Y 137.839,Z 605.581,A -85,B 0,C 180,E1 -25708.613,E2 -25708.613} C_VEL
LIN {X 0,Y 134.389,Z 604.372,A -85,B 0,C 180,E1 -25710.569,E2 -25710.569} C_VEL
LIN {X 0,Y 127.795,Z 601.741,A -85,B 0,C 180,E1 -25713.595,E2 -25713.595} C_VEL
LIN {X 0,Y 122.869,Z 599.211,A -85,B 0,C 180,E1 -25716.195,E2 -25716.195} C_VEL
LIN {X 0,Y 120.092,Z 597.192,A -85,B 0,C 180,E1 -25718.461,E2 -25718.461} C_VEL
LIN {X 0,Y 119.454,Z 596.492,A -85,B 0,C 180,E1 -25719.291,E2 -25719.291} C_VEL
LIN {X 0,Y 115.569,Z 589.504,A -85,B 0,C 180,E1 -25727.247,E2 -25727.247} C_VEL
LIN {X 0,Y 114.363,Z 582.647,A -85,B 0,C 180,E1 -25733.827,E2 -25733.827} C_VEL
LIN {X 0,Y 114.036,Z 575.304,A -85,B 0,C 180,E1 -25739.78,E2 -25739.78} C_VEL
LIN {X 0,Y 114.311,Z 575.18,A -85,B 0,C 180,E1 -25743.525,E2 -25743.525} C_VEL
LIN {X 0,Y 116.516,Z 573.241,A -85,B 0,C 180,E1 -25746.929,E2 -25746.929} C_VEL
LIN {X 0,Y 117.974,Z 572.7,A -85,B 0,C 180,E1 -25750.295,E2 -25750.295} C_VEL
LIN {X 0,Y 120.684,Z 571.026,A -85,B 0,C 180,E1 -25753.47,E2 -25753.47} C_VEL
LIN {X 0,Y 123.439,Z 569.702,A -85,B 0,C 180,E1 -25756.54,E2 -25756.54} C_VEL
LIN {X 0,Y 132.573,Z 565.107,A -85,B 0,C 180,E1 -25763.428,E2 -25763.428} C_VEL
LIN {X 0,Y 134.693,Z 563.993,A -85,B 0,C 180,E1 -25764.672,E2 -25764.672} C_VEL
LIN {X 0,Y 137.232,Z 562.303,A -85,B 0,C 180,E1 -25765.805,E2 -25765.805} C_VEL
LIN {X 0,Y 144.167,Z 558.676,A -85,B 0,C 180,E1 -25769.176,E2 -25769.176} C_VEL
LIN {X 0,Y 147.586,Z 556.479,A -85,B 0,C 180,E1 -25770.446,E2 -25770.446} C_VEL
LIN {X 0,Y 149.353,Z 555.581,A -85,B 0,C 180,E1 -25771.173,E2 -25771.173} C_VEL
LIN {X 0,Y 153.429,Z 554.914,A -85,B 0,C 180,E1 -25773.345,E2 -25773.345} C_VEL
LIN {X 0,Y 153.62,Z 557.554,A -85,B 0,C 180,E1 -25774.56,E2 -25774.56} C_VEL
LIN {X 0,Y 152.414,Z 566.686,A -85,B 0,C 180,E1 -25777.868,E2 -25777.868} C_VEL
LIN {X 0,Y 150.087,Z 576.488,A -85,B 0,C 180,E1 -25781.473,E2 -25781.473} C_VEL
LIN {X 0,Y 143.31,Z 587.362,A -85,B 0,C 180,E1 -25784.672,E2 -25784.672} C_VEL
LIN {X 0,Y 137.124,Z 596.33,A -85,B 0,C 180,E1 -25788.214,E2 -25788.214} C_VEL
LIN {X 0,Y 130.544,Z 604.894,A -85,B 0,C 180,E1 -25792.719,E2 -25792.719} C_VEL
LIN {X 0,Y 124.919,Z 611.672,A -85,B 0,C 180,E1 -25797.555,E2 -25797.555} C_VEL
LIN {X 0,Y 120.931,Z 616.567,A -85,B 0,C 180,E1 -25802.29,E2 -25802.29} C_VEL
LIN {X 0,Y 116.579,Z 621.482,A -85,B 0,C 180,E1 -25808.79,E2 -25808.79} C_VEL
LIN {X 0,Y 113.816,Z 624.901,A -85,B 0,C 180,E1 -25815.696,E2 -25815.696} C_VEL
LIN {X 0,Y 112.374,Z 626.932,A -85,B 0,C 180,E1 -25822.81,E2 -25822.81} C_VEL
LIN {X 0,Y 112.199,Z 627.622,A -85,B 0,C 180,E1 -25829.995,E2 -25829.995} C_VEL
LIN {X 0,Y 112.37,Z 626.982,A -85,B 0,C 180,E1 -25837.181,E2 -25837.181} C_VEL
LIN {X 0,Y 113.796,Z 624.994,A -85,B 0,C 180,E1 -25844.298,E2 -25844.298} C_VEL
LIN {X 0,Y 116.507,Z 621.614,A -85,B 0,C 180,E1 -25851.214,E2 -25851.214} C_VEL
LIN {X 0,Y 120.858,Z 616.737,A -85,B 0,C 180,E1 -25857.719,E2 -25857.719} C_VEL
LIN {X 0,Y 126.33,Z 610.224,A -85,B 0,C 180,E1 -25863.796,E2 -25863.796} C_VEL
LIN {X 0,Y 132.285,Z 602.95,A -85,B 0,C 180,E1 -25868.622,E2 -25868.622} C_VEL
LIN {X 0,Y 139.023,Z 593.876,A -85,B 0,C 180,E1 -25873.031,E2 -25873.031} C_VEL
LIN {X 0,Y 145.477,Z 584.379,A -85,B 0,C 180,E1 -25876.434,E2 -25876.434} C_VEL
LIN {X 0,Y 149.991,Z 576.959,A -85,B 0,C 180,E1 -25878.559,E2 -25878.559} C_VEL
LIN {X 0,Y 152.005,Z 569.483,A -85,B 0,C 180,E1 -25881.274,E2 -25881.274} C_VEL
LIN {X 0,Y 153.65,Z 558.902,A -85,B 0,C 180,E1 -25885.129,E2 -25885.129} C_VEL
LIN {X 0,Y 153.755,Z 556.788,A -85,B 0,C 180,E1 -25885.948,E2 -25885.948} C_VEL
LIN {X 0,Y 152.653,Z 549.547,A -85,B 0,C 180,E1 -25889.573,E2 -25889.573} C_VEL
LIN {X 0,Y 151.168,Z 543.492,A -85,B 0,C 180,E1 -25893.045,E2 -25893.045} C_VEL
LIN {X 0,Y 150.186,Z 540.296,A -85,B 0,C 180,E1 -25895.092,E2 -25895.092} C_VEL
LIN {X 0,Y 148.224,Z 534.937,A -85,B 0,C 180,E1 -25899.169,E2 -25899.169} C_VEL
LIN {X 0,Y 146.477,Z 530.538,A -85,B 0,C 180,E1 -25903.269,E2 -25903.269} C_VEL
LIN {X 0,Y 145.036,Z 526.904,A -85,B 0,C 180,E1 -25907.405,E2 -25907.405} C_VEL
LIN {X 0,Y 144.627,Z 525.979,A -85,B 0,C 180,E1 -25908.791,E2 -25908.791} C_VEL
LIN {X 0,Y 143.1,Z 522.959,A -85,B 0,C 180,E1 -25916.48,E2 -25916.48} C_VEL
LIN {X 0,Y 143.119,Z 521.989,A -85,B 0,C 180,E1 -25920,E2 -25920} C_VEL
LIN {X 0,Y 143.541,Z 523.52,A -85,B 0,C 180,E1 -25926.325,E2 -25926.325} C_VEL
LIN {X 0,Y 144.828,Z 525.474,A -85,B 0,C 180,E1 -25931.192,E2 -25931.192} C_VEL
LIN {X 0,Y 145.754,Z 527.278,A -85,B 0,C 180,E1 -25933.951,E2 -25933.951} C_VEL
LIN {X 0,Y 148.201,Z 532.038,A -85,B 0,C 180,E1 -25939.387,E2 -25939.387} C_VEL
LIN {X 0,Y 150.192,Z 536.197,A -85,B 0,C 180,E1 -25943.092,E2 -25943.092} C_VEL
LIN {X 0,Y 152.6,Z 542.465,A -85,B 0,C 180,E1 -25947.422,E2 -25947.422} C_VEL
LIN {X 0,Y 154.488,Z 548.1,A -85,B 0,C 180,E1 -25950.783,E2 -25950.783} C_VEL
LIN {X 0,Y 155.654,Z 556.409,A -85,B 0,C 180,E1 -25954.565,E2 -25954.565} C_VEL
LIN {X 0,Y 155.882,Z 560.467,A -85,B 0,C 180,E1 -25956.28,E2 -25956.28} C_VEL
LIN {X 0,Y 153.379,Z 569.431,A -85,B 0,C 180,E1 -25958.84,E2 -25958.84} C_VEL
LIN {X 0,Y 151.833,Z 573.98,A -85,B 0,C 180,E1 -25960.212,E2 -25960.212} C_VEL
LIN {X 0,Y 146.187,Z 583.912,A -85,B 0,C 180,E1 -25962.854,E2 -25962.854} C_VEL
LIN {X 0,Y 139.628,Z 593.789,A -85,B 0,C 180,E1 -25966.21,E2 -25966.21} C_VEL
LIN {X 0,Y 133.645,Z 601.98,A -85,B 0,C 180,E1 -25969.9,E2 -25969.9} C_VEL
LIN {X 0,Y 127.43,Z 609.802,A -85,B 0,C 180,E1 -25974.618,E2 -25974.618} C_VEL
LIN {X 0,Y 122.635,Z 615.539,A -85,B 0,C 180,E1 -25979.274,E2 -25979.274} C_VEL
LIN {X 0,Y 118.158,Z 621.004,A -85,B 0,C 180,E1 -25985.4,E2 -25985.4} C_VEL
LIN {X 0,Y 114.634,Z 625.164,A -85,B 0,C 180,E1 -25992.154,E2 -25992.154} C_VEL
LIN {X 0,Y 112.733,Z 627.878,A -85,B 0,C 180,E1 -25999.225,E2 -25999.225} C_VEL
LIN {X 0,Y 112.113,Z 629.22,A -85,B 0,C 180,E1 -26006.411,E2 -26006.411} C_VEL
LIN {X 0,Y 112.198,Z 629.384,A -85,B 0,C 180,E1 -26010.005,E2 -26010.005} C_VEL
LIN {X 0,Y 112.266,Z 628.688,A -85,B 0,C 180,E1 -26017.197,E2 -26017.197} C_VEL
LIN {X 0,Y 113.524,Z 626.639,A -85,B 0,C 180,E1 -26024.342,E2 -26024.342} C_VEL
LIN {X 0,Y 116.201,Z 623.191,A -85,B 0,C 180,E1 -26031.282,E2 -26031.282} C_VEL
LIN {X 0,Y 120.481,Z 618.242,A -85,B 0,C 180,E1 -26037.822,E2 -26037.822} C_VEL
LIN {X 0,Y 124.741,Z 613.396,A -85,B 0,C 180,E1 -26042.41,E2 -26042.41} C_VEL
LIN {X 0,Y 129.829,Z 608.119,A -85,B 0,C 180,E1 -26046.309,E2 -26046.309} C_VEL
LIN {X 0,Y 137.882,Z 609.183,A -85,B 0,C 180,E1 -26051.505,E2 -26051.505} C_VEL
LIN {X 0,Y 149.946,Z 609.423,A -85,B 0,C 180,E1 -26057.018,E2 -26057.018} C_VEL
LIN {X 0,Y 149.738,Z 609.25,A -85,B 0,C 180,E1 -26057.926,E2 -26057.926} C_VEL
LIN {X 0,Y 139.14,Z 607.351,A -85,B 0,C 180,E1 -26062.69,E2 -26062.69} C_VEL
LIN {X 0,Y 131.042,Z 604.67,A -85,B 0,C 180,E1 -26067.567,E2 -26067.567} C_VEL
LIN {X 0,Y 124.424,Z 601.059,A -85,B 0,C 180,E1 -26073.136,E2 -26073.136} C_VEL
LIN {X 0,Y 119.454,Z 596.492,A -85,B 0,C 180,E1 -26079.291,E2 -26079.291} C_VEL
LIN {X 0,Y 117.794,Z 594.984,A -85,B 0,C 180,E1 -26080.874,E2 -26080.874} C_VEL
LIN {X 0,Y 113.743,Z 592.03,A -85,B 0,C 180,E1 -26083.111,E2 -26083.111} C_VEL
LIN {X 0,Y 109.932,Z 588.812,A -85,B 0,C 180,E1 -26085.458,E2 -26085.458} C_VEL
LIN {X 0,Y 108.728,Z 586.89,A -85,B 0,C 180,E1 -26087.186,E2 -26087.186} C_VEL
LIN {X 0,Y 107.923,Z 583.713,A -85,B 0,C 180,E1 -26090.631,E2 -26090.631} C_VEL
LIN {X 0,Y 107.417,Z 583.685,A -85,B 0,C 180,E1 -26092.481,E2 -26092.481} C_VEL
LIN {X 0,Y 107.615,Z 582.757,A -85,B 0,C 180,E1 -26096.256,E2 -26096.256} C_VEL
LIN {X 0,Y 109.044,Z 580.95,A -85,B 0,C 180,E1 -26100,E2 -26100} C_VEL
LIN {X 0,Y 109.639,Z 580.494,A -85,B 0,C 180,E1 -26103.676,E2 -26103.676} C_VEL
LIN {X 0,Y 111.667,Z 578.944,A -85,B 0,C 180,E1 -26107.232,E2 -26107.232} C_VEL
LIN {X 0,Y 113.445,Z 578.137,A -85,B 0,C 180,E1 -26110.711,E2 -26110.711} C_VEL
LIN {X 0,Y 122.505,Z 573.822,A -85,B 0,C 180,E1 -26120.134,E2 -26120.134} C_VEL
LIN {X 0,Y 132.952,Z 568.952,A -85,B 0,C 180,E1 -26126.702,E2 -26126.702} C_VEL
LIN {X 0,Y 135.622,Z 567.354,A -85,B 0,C 180,E1 -26127.8,E2 -26127.8} C_VEL
LIN {X 0,Y 143.404,Z 563.531,A -85,B 0,C 180,E1 -26131.223,E2 -26131.223} C_VEL
LIN {X 0,Y 145.783,Z 562.117,A -85,B 0,C 180,E1 -26132.026,E2 -26132.026} C_VEL
LIN {X 0,Y 148.154,Z 561.269,A -85,B 0,C 180,E1 -26133.061,E2 -26133.061} C_VEL
LIN {X 0,Y 148.331,Z 562.629,A -85,B 0,C 180,E1 -26133.83,E2 -26133.83} C_VEL
LIN {X 0,Y 146.313,Z 572.355,A -85,B 0,C 180,E1 -26137.572,E2 -26137.572} C_VEL
LIN {X 0,Y 144.672,Z 577.827,A -85,B 0,C 180,E1 -26139.714,E2 -26139.714} C_VEL
LIN {X 0,Y 138.411,Z 587.414,A -85,B 0,C 180,E1 -26142.582,E2 -26142.582} C_VEL
LIN {X 0,Y 131.892,Z 596.384,A -85,B 0,C 180,E1 -26146.149,E2 -26146.149} C_VEL
LIN {X 0,Y 124.957,Z 604.949,A -85,B 0,C 180,E1 -26150.743,E2 -26150.743} C_VEL
LIN {X 0,Y 118.56,Z 612.172,A -85,B 0,C 180,E1 -26156.089,E2 -26156.089} C_VEL
LIN {X 0,Y 113.389,Z 618.03,A -85,B 0,C 180,E1 -26162.294,E2 -26162.294} C_VEL
LIN {X 0,Y 109.96,Z 621.538,A -85,B 0,C 180,E1 -26167.445,E2 -26167.445} C_VEL
LIN {X 0,Y 106.927,Z 624.958,A -85,B 0,C 180,E1 -26174.752,E2 -26174.752} C_VEL
LIN {X 0,Y 105.319,Z 626.988,A -85,B 0,C 180,E1 -26182.326,E2 -26182.326} C_VEL
LIN {X 0,Y 105.106,Z 627.678,A -85,B 0,C 180,E1 -26189.995,E2 -26189.995} C_VEL
LIN {X 0,Y 105.315,Z 627.037,A -85,B 0,C 180,E1 -26197.665,E2 -26197.665} C_VEL
LIN {X 0,Y 106.906,Z 625.049,A -85,B 0,C 180,E1 -26205.241,E2 -26205.241} C_VEL
LIN {X 0,Y 109.888,Z 621.668,A -85,B 0,C 180,E1 -26212.56,E2 -26212.56} C_VEL
LIN {X 0,Y 114.574,Z 616.791,A -85,B 0,C 180,E1 -26219.383,E2 -26219.383} C_VEL
LIN {X 0,Y 120.457,Z 610.276,A -85,B 0,C 180,E1 -26225.688,E2 -26225.688} C_VEL
LIN {X 0,Y 126.809,Z 603.001,A -85,B 0,C 180,E1 -26230.627,E2 -26230.627} C_VEL
LIN {X 0,Y 133.907,Z 593.925,A -85,B 0,C 180,E1 -26235.11,E2 -26235.11} C_VEL
LIN {X 0,Y 140.658,Z 584.425,A -85,B 0,C 180,E1 -26238.539,E2 -26238.539} C_VEL
LIN {X 0,Y 144.642,Z 578.176,A -85,B 0,C 180,E1 -26240.35,E2 -26240.35} C_VEL
LIN {X 0,Y 146.645,Z 571.798,A -85,B 0,C 180,E1 -26242.814,E2 -26242.814} C_VEL
LIN {X 0,Y 148.594,Z 561.896,A -85,B 0,C 180,E1 -26246.646,E2 -26246.646} C_VEL
LIN {X 0,Y 148.546,Z 558.261,A -85,B 0,C 180,E1 -26248.38,E2 -26248.38} C_VEL
LIN {X 0,Y 147.522,Z 551.333,A -85,B 0,C 180,E1 -26252.322,E2 -26252.322} C_VEL
LIN {X 0,Y 146.31,Z 545.941,A -85,B 0,C 180,E1 -26255.866,E2 -26255.866} C_VEL
LIN {X 0,Y 144.707,Z 540.633,A -85,B 0,C 180,E1 -26260.125,E2 -26260.125} C_VEL
LIN {X 0,Y 143.418,Z 536.667,A -85,B 0,C 180,E1 -26263.999,E2 -26263.999} C_VEL
LIN {X 0,Y 142.183,Z 532.896,A -85,B 0,C 180,E1 -26268.596,E2 -26268.596} C_VEL
LIN {X 0,Y 141.047,Z 530.393,A -85,B 0,C 180,E1 -26274.28,E2 -26274.28} C_VEL
LIN {X 0,Y 140.917,Z 528.766,A -85,B 0,C 180,E1 -26280,E2 -26280} C_VEL
LIN {X 0,Y 141.17,Z 530.088,A -85,B 0,C 180,E1 -26285.714,E2 -26285.714} C_VEL
LIN {X 0,Y 142.431,Z 532.409,A -85,B 0,C 180,E1 -26291.383,E2 -26291.383} C_VEL
LIN {X 0,Y 144.88,Z 537.832,A -85,B 0,C 180,E1 -26298.379,E2 -26298.379} C_VEL
LIN {X 0,Y 146.718,Z 542.269,A -85,B 0,C 180,E1 -26302.532,E2 -26302.532} C_VEL
LIN {X 0,Y 148.947,Z 548.99,A -85,B 0,C 180,E1 -26307.389,E2 -26307.389} C_VEL
LIN {X 0,Y 150.118,Z 554.114,A -85,B 0,C 180,E1 -26310.419,E2 -26310.419} C_VEL
LIN {X 0,Y 150.712,Z 562.628,A -85,B 0,C 180,E1 -26314.476,E2 -26314.476} C_VEL
LIN {X 0,Y 150.555,Z 563.894,A -85,B 0,C 180,E1 -26314.97,E2 -26314.97} C_VEL
LIN {X 0,Y 147.125,Z 573.935,A -85,B 0,C 180,E1 -26317.992,E2 -26317.992} C_VEL
LIN {X 0,Y 146.137,Z 576.056,A -85,B 0,C 180,E1 -26318.611,E2 -26318.611} C_VEL
LIN {X 0,Y 140.253,Z 585.633,A -85,B 0,C 180,E1 -26321.273,E2 -26321.273} C_VEL
LIN {X 0,Y 133.467,Z 595.216,A -85,B 0,C 180,E1 -26324.7,E2 -26324.7} C_VEL
LIN {X 0,Y 127.28,Z 603.153,A -85,B 0,C 180,E1 -26328.507,E2 -26328.507} C_VEL
LIN {X 0,Y 121.692,Z 609.75,A -85,B 0,C 180,E1 -26332.676,E2 -26332.676} C_VEL
LIN {X 0,Y 115.611,Z 616.575,A -85,B 0,C 180,E1 -26338.575,E2 -26338.575} C_VEL
LIN {X 0,Y 111.676,Z 620.95,A -85,B 0,C 180,E1 -26343.868,E2 -26343.868} C_VEL
LIN {X 0,Y 107.853,Z 625.109,A -85,B 0,C 180,E1 -26350.99,E2 -26350.99} C_VEL
LIN {X 0,Y 105.753,Z 627.823,A -85,B 0,C 180,E1 -26358.505,E2 -26358.505} C_VEL
LIN {X 0,Y 105.025,Z 629.165,A -85,B 0,C 180,E1 -26366.168,E2 -26366.168} C_VEL
LIN {X 0,Y 105.104,Z 629.328,A -85,B 0,C 180,E1 -26370.005,E2 -26370.005} C_VEL
LIN {X 0,Y 105.222,Z 628.632,A -85,B 0,C 180,E1 -26377.682,E2 -26377.682} C_VEL
LIN {X 0,Y 106.61,Z 626.583,A -85,B 0,C 180,E1 -26385.294,E2 -26385.294} C_VEL
LIN {X 0,Y 109.597,Z 623.135,A -85,B 0,C 180,E1 -26392.633,E2 -26392.633} C_VEL
LIN {X 0,Y 114.23,Z 618.186,A -85,B 0,C 180,E1 -26399.49,E2 -26399.49} C_VEL
LIN {X 0,Y 118.755,Z 613.385,A -85,B 0,C 180,E1 -26404.212,E2 -26404.212} C_VEL
LIN {X 0,Y 125.243,Z 606.905,A -85,B 0,C 180,E1 -26408.892,E2 -26408.892} C_VEL
LIN {X 0,Y 137.288,Z 608.458,A -85,B 0,C 180,E1 -26415.786,E2 -26415.786} C_VEL
LIN {X 0,Y 140.025,Z 608.593,A -85,B 0,C 180,E1 -26416.992,E2 -26416.992} C_VEL
LIN {X 0,Y 139.646,Z 608.361,A -85,B 0,C 180,E1 -26417.984,E2 -26417.984} C_VEL
LIN {X 0,Y 129.238,Z 605.502,A -85,B 0,C 180,E1 -26423.26,E2 -26423.26} C_VEL
LIN {X 0,Y 119.757,Z 601.012,A -85,B 0,C 180,E1 -26430.078,E2 -26430.078} C_VEL
LIN {X 0,Y 112.979,Z 594.976,A -85,B 0,C 180,E1 -26438.085,E2 -26438.085} C_VEL
LIN {X 0,Y 109.359,Z 588.848,A -85,B 0,C 180,E1 -26445.105,E2 -26445.105} C_VEL
LIN {X 0,Y 108.728,Z 586.89,A -85,B 0,C 180,E1 -26447.186,E2 -26447.186} C_VEL
LIN {X 0,Y 107.947,Z 585.932,A -85,B 0,C 180,E1 -26448.792,E2 -26448.792} C_VEL
LIN {X 0,Y 106.186,Z 585.912,A -85,B 0,C 180,E1 -26451.125,E2 -26451.125} C_VEL
LIN {X 0,Y 103.143,Z 587.252,A -85,B 0,C 180,E1 -26456.065,E2 -26456.065} C_VEL
LIN {X 0,Y 103.14,Z 587.045,A -85,B 0,C 180,E1 -26458.206,E2 -26458.206} C_VEL
LIN {X 0,Y 103.169,Z 586.987,A -85,B 0,C 180,E1 -26458.297,E2 -26458.297} C_VEL
LIN {X 0,Y 103.792,Z 586.327,A -85,B 0,C 180,E1 -26460,E2 -26460} C_VEL
LIN {X 0,Y 104.711,Z 585.591,A -85,B 0,C 180,E1 -26463.849,E2 -26463.849} C_VEL
LIN {X 0,Y 106.631,Z 584.311,A -85,B 0,C 180,E1 -26467.575,E2 -26467.575} C_VEL
LIN {X 0,Y 111.329,Z 582.18,A -85,B 0,C 180,E1 -26474.627,E2 -26474.627} C_VEL
LIN {X 0,Y 117.991,Z 579.38,A -85,B 0,C 180,E1 -26480.94,E2 -26480.94} C_VEL
LIN {X 0,Y 128.688,Z 574.944,A -85,B 0,C 180,E1 -26487.659,E2 -26487.659} C_VEL
LIN {X 0,Y 131.187,Z 573.78,A -85,B 0,C 180,E1 -26488.826,E2 -26488.826} C_VEL
LIN {X 0,Y 133.991,Z 572.266,A -85,B 0,C 180,E1 -26489.887,E2 -26489.887} C_VEL
LIN {X 0,Y 141.787,Z 568.722,A -85,B 0,C 180,E1 -26493.041,E2 -26493.041} C_VEL
LIN {X 0,Y 142.465,Z 569.083,A -85,B 0,C 180,E1 -26493.664,E2 -26493.664} C_VEL
LIN {X 0,Y 140.142,Z 577.187,A -85,B 0,C 180,E1 -26496.999,E2 -26496.999} C_VEL
LIN {X 0,Y 139.453,Z 579.055,A -85,B 0,C 180,E1 -26497.785,E2 -26497.785} C_VEL
LIN {X 0,Y 132.507,Z 589.074,A -85,B 0,C 180,E1 -26500.899,E2 -26500.899} C_VEL
LIN {X 0,Y 125.773,Z 597.776,A -85,B 0,C 180,E1 -26504.56,E2 -26504.56} C_VEL
LIN {X 0,Y 118.545,Z 606.108,A -85,B 0,C 180,E1 -26509.292,E2 -26509.292} C_VEL
LIN {X 0,Y 112.397,Z 612.575,A -85,B 0,C 180,E1 -26514.378,E2 -26514.378} C_VEL
LIN {X 0,Y 107.124,Z 618.086,A -85,B 0,C 180,E1 -26520.52,E2 -26520.52} C_VEL
LIN {X 0,Y 103.413,Z 621.594,A -85,B 0,C 180,E1 -26525.931,E2 -26525.931} C_VEL
LIN {X 0,Y 100.078,Z 625.014,A -85,B 0,C 180,E1 -26533.681,E2 -26533.681} C_VEL
LIN {X 0,Y 98.288,Z 627.044,A -85,B 0,C 180,E1 -26541.773,E2 -26541.773} C_VEL
LIN {X 0,Y 98.006,Z 627.734,A -85,B 0,C 180,E1 -26549.995,E2 -26549.995} C_VEL
LIN {X 0,Y 98.285,Z 627.093,A -85,B 0,C 180,E1 -26558.217,E2 -26558.217} C_VEL
LIN {X 0,Y 100.057,Z 625.104,A -85,B 0,C 180,E1 -26566.312,E2 -26566.312} C_VEL
LIN {X 0,Y 103.346,Z 621.723,A -85,B 0,C 180,E1 -26574.075,E2 -26574.075} C_VEL
LIN {X 0,Y 108.403,Z 616.845,A -85,B 0,C 180,E1 -26581.236,E2 -26581.236} C_VEL
LIN {X 0,Y 114.738,Z 610.329,A -85,B 0,C 180,E1 -26587.766,E2 -26587.766} C_VEL
LIN {X 0,Y 121.497,Z 603.052,A -85,B 0,C 180,E1 -26592.812,E2 -26592.812} C_VEL
LIN {X 0,Y 128.97,Z 593.974,A -85,B 0,C 180,E1 -26597.356,E2 -26597.356} C_VEL
LIN {X 0,Y 136.053,Z 584.471,A -85,B 0,C 180,E1 -26600.784,E2 -26600.784} C_VEL
LIN {X 0,Y 139.493,Z 579.339,A -85,B 0,C 180,E1 -26602.284,E2 -26602.284} C_VEL
LIN {X 0,Y 141.931,Z 571.913,A -85,B 0,C 180,E1 -26605.36,E2 -26605.36} C_VEL
LIN {X 0,Y 143.593,Z 564.787,A -85,B 0,C 180,E1 -26608.28,E2 -26608.28} C_VEL
LIN {X 0,Y 143.536,Z 560.438,A -85,B 0,C 180,E1 -26610.683,E2 -26610.683} C_VEL
LIN {X 0,Y 142.63,Z 553.431,A -85,B 0,C 180,E1 -26615.202,E2 -26615.202} C_VEL
LIN {X 0,Y 141.418,Z 547.832,A -85,B 0,C 180,E1 -26619.642,E2 -26619.642} C_VEL
LIN {X 0,Y 140.319,Z 543.312,A -85,B 0,C 180,E1 -26624.01,E2 -26624.01} C_VEL
LIN {X 0,Y 139.348,Z 539.832,A -85,B 0,C 180,E1 -26628.361,E2 -26628.361} C_VEL
LIN {X 0,Y 138.822,Z 538.24,A -85,B 0,C 180,E1 -26631.264,E2 -26631.264} C_VEL
LIN {X 0,Y 138.256,Z 536.217,A -85,B 0,C 180,E1 -26637.086,E2 -26637.086} C_VEL
LIN {X 0,Y 138.389,Z 535.451,A -85,B 0,C 180,E1 -26640,E2 -26640} C_VEL
LIN {X 0,Y 138.59,Z 536.784,A -85,B 0,C 180,E1 -26645.821,E2 -26645.821} C_VEL
LIN {X 0,Y 139.069,Z 537.818,A -85,B 0,C 180,E1 -26648.72,E2 -26648.72} C_VEL
LIN {X 0,Y 140.017,Z 540.227,A -85,B 0,C 180,E1 -26653.054,E2 -26653.054} C_VEL
LIN {X 0,Y 141.368,Z 543.52,A -85,B 0,C 180,E1 -26657.354,E2 -26657.354} C_VEL
LIN {X 0,Y 142.882,Z 547.824,A -85,B 0,C 180,E1 -26661.646,E2 -26661.646} C_VEL
LIN {X 0,Y 144.684,Z 554.412,A -85,B 0,C 180,E1 -26666.7,E2 -26666.7} C_VEL
LIN {X 0,Y 145.35,Z 557.842,A -85,B 0,C 180,E1 -26668.916,E2 -26668.916} C_VEL
LIN {X 0,Y 145.529,Z 565.639,A -85,B 0,C 180,E1 -26672.932,E2 -26672.932} C_VEL
LIN {X 0,Y 144.882,Z 568.18,A -85,B 0,C 180,E1 -26673.836,E2 -26673.836} C_VEL
LIN {X 0,Y 141.757,Z 576.008,A -85,B 0,C 180,E1 -26676.335,E2 -26676.335} C_VEL
LIN {X 0,Y 135.657,Z 585.587,A -85,B 0,C 180,E1 -26679.01,E2 -26679.01} C_VEL
LIN {X 0,Y 128.568,Z 595.167,A -85,B 0,C 180,E1 -26682.449,E2 -26682.449} C_VEL
LIN {X 0,Y 122.029,Z 603.103,A -85,B 0,C 180,E1 -26686.288,E2 -26686.288} C_VEL
LIN {X 0,Y 116.095,Z 609.698,A -85,B 0,C 180,E1 -26690.539,E2 -26690.539} C_VEL
LIN {X 0,Y 109.829,Z 616.212,A -85,B 0,C 180,E1 -26696.291,E2 -26696.291} C_VEL
LIN {X 0,Y 105.289,Z 620.895,A -85,B 0,C 180,E1 -26702.15,E2 -26702.15} C_VEL
LIN {X 0,Y 101.124,Z 625.054,A -85,B 0,C 180,E1 -26709.671,E2 -26709.671} C_VEL
LIN {X 0,Y 98.768,Z 627.768,A -85,B 0,C 180,E1 -26717.68,E2 -26717.68} C_VEL
LIN {X 0,Y 97.934,Z 629.109,A -85,B 0,C 180,E1 -26725.89,E2 -26725.89} C_VEL
LIN {X 0,Y 98.004,Z 629.272,A -85,B 0,C 180,E1 -26730.005,E2 -26730.005} C_VEL
LIN {X 0,Y 98.178,Z 628.576,A -85,B 0,C 180,E1 -26738.236,E2 -26738.236} C_VEL
LIN {X 0,Y 99.738,Z 626.527,A -85,B 0,C 180,E1 -26746.376,E2 -26746.376} C_VEL
LIN {X 0,Y 103.036,Z 623.079,A -85,B 0,C 180,E1 -26754.163,E2 -26754.163} C_VEL
LIN {X 0,Y 108.087,Z 618.13,A -85,B 0,C 180,E1 -26761.349,E2 -26761.349} C_VEL
LIN {X 0,Y 112.764,Z 613.508,A -85,B 0,C 180,E1 -26766.089,E2 -26766.089} C_VEL
LIN {X 0,Y 120.061,Z 606.39,A -85,B 0,C 180,E1 -26771.194,E2 -26771.194} C_VEL
LIN {X 0,Y 121.079,Z 605.551,A -85,B 0,C 180,E1 -26771.741,E2 -26771.741} C_VEL
LIN {X 0,Y 130.343,Z 607.075,A -85,B 0,C 180,E1 -26776.957,E2 -26776.957} C_VEL
LIN {X 0,Y 129.782,Z 606.742,A -85,B 0,C 180,E1 -26778.077,E2 -26778.077} C_VEL
LIN {X 0,Y 119.415,Z 602.886,A -85,B 0,C 180,E1 -26783.947,E2 -26783.947} C_VEL
LIN {X 0,Y 112.15,Z 598.59,A -85,B 0,C 180,E1 -26789.912,E2 -26789.912} C_VEL
LIN {X 0,Y 106.047,Z 592.555,A -85,B 0,C 180,E1 -26797.6,E2 -26797.6} C_VEL
LIN {X 0,Y 105.517,Z 591.806,A -85,B 0,C 180,E1 -26798.511,E2 -26798.511} C_VEL
LIN {X 0,Y 103.377,Z 591.561,A -85,B 0,C 180,E1 -26802.148,E2 -26802.148} C_VEL
LIN {X 0,Y 102.755,Z 591.138,A -85,B 0,C 180,E1 -26804.123,E2 -26804.123} C_VEL
LIN {X 0,Y 102.395,Z 588.657,A -85,B 0,C 180,E1 -26812.11,E2 -26812.11} C_VEL
LIN {X 0,Y 102.502,Z 587.839,A -85,B 0,C 180,E1 -26816.069,E2 -26816.069} C_VEL
LIN {X 0,Y 103.169,Z 586.987,A -85,B 0,C 180,E1 -26818.297,E2 -26818.297} C_VEL
LIN {X 0,Y 103.766,Z 586.375,A -85,B 0,C 180,E1 -26821.516,E2 -26821.516} C_VEL
LIN {X 0,Y 103.788,Z 586.996,A -85,B 0,C 180,E1 -26826.983,E2 -26826.983} C_VEL
LIN {X 0,Y 104.641,Z 587.71,A -85,B 0,C 180,E1 -26832.434,E2 -26832.434} C_VEL
LIN {X 0,Y 106.473,Z 587.254,A -85,B 0,C 180,E1 -26835.478,E2 -26835.478} C_VEL
LIN {X 0,Y 117.399,Z 583.16,A -85,B 0,C 180,E1 -26844.775,E2 -26844.775} C_VEL
LIN {X 0,Y 126.777,Z 579.589,A -85,B 0,C 180,E1 -26849.929,E2 -26849.929} C_VEL
LIN {X 0,Y 135.012,Z 575.942,A -85,B 0,C 180,E1 -26853.126,E2 -26853.126} C_VEL
LIN {X 0,Y 135.803,Z 576.653,A -85,B 0,C 180,E1 -26854.098,E2 -26854.098} C_VEL
LIN {X 0,Y 134.392,Z 580.263,A -85,B 0,C 180,E1 -26855.686,E2 -26855.686} C_VEL
LIN {X 0,Y 127.97,Z 589.126,A -85,B 0,C 180,E1 -26858.495,E2 -26858.495} C_VEL
LIN {X 0,Y 120.871,Z 597.83,A -85,B 0,C 180,E1 -26862.148,E2 -26862.148} C_VEL
LIN {X 0,Y 114.287,Z 605.059,A -85,B 0,C 180,E1 -26866.221,E2 -26866.221} C_VEL
LIN {X 0,Y 107.363,Z 611.965,A -85,B 0,C 180,E1 -26871.544,E2 -26871.544} C_VEL
LIN {X 0,Y 100.973,Z 618.142,A -85,B 0,C 180,E1 -26878.526,E2 -26878.526} C_VEL
LIN {X 0,Y 96.955,Z 621.65,A -85,B 0,C 180,E1 -26884.214,E2 -26884.214} C_VEL
LIN {X 0,Y 93.26,Z 625.07,A -85,B 0,C 180,E1 -26892.451,E2 -26892.451} C_VEL
LIN {X 0,Y 91.258,Z 627.1,A -85,B 0,C 180,E1 -26901.134,E2 -26901.134} C_VEL
LIN {X 0,Y 90.914,Z 627.79,A -85,B 0,C 180,E1 -26909.994,E2 -26909.994} C_VEL
LIN {X 0,Y 91.254,Z 627.148,A -85,B 0,C 180,E1 -26918.855,E2 -26918.855} C_VEL
LIN {X 0,Y 93.236,Z 625.159,A -85,B 0,C 180,E1 -26927.543,E2 -26927.543} C_VEL
LIN {X 0,Y 96.891,Z 621.777,A -85,B 0,C 180,E1 -26935.793,E2 -26935.793} C_VEL
LIN {X 0,Y 100.916,Z 618.298,A -85,B 0,C 180,E1 -26941.482,E2 -26941.482} C_VEL
LIN {X 0,Y 107.347,Z 612.172,A -85,B 0,C 180,E1 -26948.451,E2 -26948.451} C_VEL
LIN {X 0,Y 114.219,Z 605.317,A -85,B 0,C 180,E1 -26953.8,E2 -26953.8} C_VEL
LIN {X 0,Y 121.953,Z 596.802,A -85,B 0,C 180,E1 -26958.512,E2 -26958.512} C_VEL
LIN {X 0,Y 129.185,Z 587.891,A -85,B 0,C 180,E1 -26962.07,E2 -26962.07} C_VEL
LIN {X 0,Y 134.443,Z 580.566,A -85,B 0,C 180,E1 -26964.365,E2 -26964.365} C_VEL
LIN {X 0,Y 136.936,Z 573.696,A -85,B 0,C 180,E1 -26967.368,E2 -26967.368} C_VEL
LIN {X 0,Y 138.458,Z 568.471,A -85,B 0,C 180,E1 -26969.636,E2 -26969.636} C_VEL
LIN {X 0,Y 138.626,Z 564.495,A -85,B 0,C 180,E1 -26971.989,E2 -26971.989} C_VEL
LIN {X 0,Y 138.212,Z 558.375,A -85,B 0,C 180,E1 -26976.237,E2 -26976.237} C_VEL
LIN {X 0,Y 137.397,Z 552.996,A -85,B 0,C 180,E1 -26980.81,E2 -26980.81} C_VEL
LIN {X 0,Y 136.661,Z 548.916,A -85,B 0,C 180,E1 -26985.1,E2 -26985.1} C_VEL
LIN {X 0,Y 136.095,Z 546.082,A -85,B 0,C 180,E1 -26988.842,E2 -26988.842} C_VEL
LIN {X 0,Y 135.8,Z 544.855,A -85,B 0,C 180,E1 -26991.068,E2 -26991.068} C_VEL
LIN {X 0,Y 135.374,Z 542.768,A -85,B 0,C 180,E1 -26997.024,E2 -26997.024} C_VEL
LIN {X 0,Y 135.55,Z 541.998,A -85,B 0,C 180,E1 -27000,E2 -27000} C_VEL
LIN {X 0,Y 135.701,Z 543.333,A -85,B 0,C 180,E1 -27005.945,E2 -27005.945} C_VEL
LIN {X 0,Y 136.097,Z 544.434,A -85,B 0,C 180,E1 -27008.912,E2 -27008.912} C_VEL
LIN {X 0,Y 136.724,Z 546.312,A -85,B 0,C 180,E1 -27012.424,E2 -27012.424} C_VEL
LIN {X 0,Y 138.04,Z 550.428,A -85,B 0,C 180,E1 -27017.787,E2 -27017.787} C_VEL
LIN {X 0,Y 138.866,Z 553.268,A -85,B 0,C 180,E1 -27020.749,E2 -27020.749} C_VEL
LIN {X 0,Y 140.075,Z 558.969,A -85,B 0,C 180,E1 -27025.439,E2 -27025.439} C_VEL
LIN {X 0,Y 140.582,Z 561.924,A -85,B 0,C 180,E1 -27027.544,E2 -27027.544} C_VEL
LIN {X 0,Y 140.464,Z 567.812,A -85,B 0,C 180,E1 -27030.854,E2 -27030.854} C_VEL
LIN {X 0,Y 140.083,Z 569.945,A -85,B 0,C 180,E1 -27031.859,E2 -27031.859} C_VEL
LIN {X 0,Y 136.407,Z 578.06,A -85,B 0,C 180,E1 -27034.484,E2 -27034.484} C_VEL
LIN {X 0,Y 130.051,Z 587.307,A -85,B 0,C 180,E1 -27037.154,E2 -27037.154} C_VEL
LIN {X 0,Y 122.666,Z 596.575,A -85,B 0,C 180,E1 -27040.618,E2 -27040.618} C_VEL
LIN {X 0,Y 115.871,Z 604.271,A -85,B 0,C 180,E1 -27044.553,E2 -27044.553} C_VEL
LIN {X 0,Y 108.721,Z 611.609,A -85,B 0,C 180,E1 -27049.734,E2 -27049.734} C_VEL
LIN {X 0,Y 103.566,Z 616.543,A -85,B 0,C 180,E1 -27054.52,E2 -27054.52} C_VEL
LIN {X 0,Y 99.014,Z 620.841,A -85,B 0,C 180,E1 -27060.214,E2 -27060.214} C_VEL
LIN {X 0,Y 94.459,Z 624.999,A -85,B 0,C 180,E1 -27068.166,E2 -27068.166} C_VEL
LIN {X 0,Y 91.817,Z 627.712,A -85,B 0,C 180,E1 -27076.731,E2 -27076.731} C_VEL
LIN {X 0,Y 90.836,Z 629.054,A -85,B 0,C 180,E1 -27085.568,E2 -27085.568} C_VEL
LIN {X 0,Y 90.911,Z 629.217,A -85,B 0,C 180,E1 -27090.006,E2 -27090.006} C_VEL
LIN {X 0,Y 91.137,Z 628.52,A -85,B 0,C 180,E1 -27098.878,E2 -27098.878} C_VEL
LIN {X 0,Y 92.916,Z 626.47,A -85,B 0,C 180,E1 -27107.617,E2 -27107.617} C_VEL
LIN {X 0,Y 96.566,Z 623.022,A -85,B 0,C 180,E1 -27115.897,E2 -27115.897} C_VEL
LIN {X 0,Y 102.074,Z 618.075,A -85,B 0,C 180,E1 -27123.429,E2 -27123.429} C_VEL
LIN {X 0,Y 107.311,Z 613.273,A -85,B 0,C 180,E1 -27128.48,E2 -27128.48} C_VEL
LIN {X 0,Y 114.828,Z 606.336,A -85,B 0,C 180,E1 -27133.521,E2 -27133.521} C_VEL
LIN {X 0,Y 117.376,Z 604.107,A -85,B 0,C 180,E1 -27134.869,E2 -27134.869} C_VEL
LIN {X 0,Y 120.032,Z 604.684,A -85,B 0,C 180,E1 -27136.404,E2 -27136.404} C_VEL
LIN {X 0,Y 121.036,Z 604.732,A -85,B 0,C 180,E1 -27137.695,E2 -27137.695} C_VEL
LIN {X 0,Y 109.762,Z 599.501,A -85,B 0,C 180,E1 -27144.812,E2 -27144.812} C_VEL
LIN {X 0,Y 108.353,Z 598.755,A -85,B 0,C 180,E1 -27145.983,E2 -27145.983} C_VEL
LIN {X 0,Y 106.059,Z 598.631,A -85,B 0,C 180,E1 -27147.987,E2 -27147.987} C_VEL
LIN {X 0,Y 103.069,Z 598.089,A -85,B 0,C 180,E1 -27151.49,E2 -27151.49} C_VEL
LIN {X 0,Y 99.195,Z 596.306,A -85,B 0,C 180,E1 -27159.253,E2 -27159.253} C_VEL
LIN {X 0,Y 97.492,Z 595.782,A -85,B 0,C 180,E1 -27163.241,E2 -27163.241} C_VEL
LIN {X 0,Y 97.001,Z 593.477,A -85,B 0,C 180,E1 -27171.668,E2 -27171.668} C_VEL
LIN {X 0,Y 97.161,Z 592.646,A -85,B 0,C 180,E1 -27175.852,E2 -27175.852} C_VEL
LIN {X 0,Y 98.4,Z 591.324,A -85,B 0,C 180,E1 -27180.104,E2 -27180.104} C_VEL
LIN {X 0,Y 103.594,Z 588.397,A -85,B 0,C 180,E1 -27191.744,E2 -27191.744} C_VEL
LIN {X 0,Y 106.473,Z 587.254,A -85,B 0,C 180,E1 -27195.478,E2 -27195.478} C_VEL
LIN {X 0,Y 108.717,Z 586.689,A -85,B 0,C 180,E1 -27198.376,E2 -27198.376} C_VEL
LIN {X 0,Y 115.27,Z 586.886,A -85,B 0,C 180,E1 -27206.86,E2 -27206.86} C_VEL
LIN {X 0,Y 118.498,Z 586.297,A -85,B 0,C 180,E1 -27209.24,E2 -27209.24} C_VEL
LIN {X 0,Y 119.763,Z 585.879,A -85,B 0,C 180,E1 -27209.929,E2 -27209.929} C_VEL
LIN {X 0,Y 124.536,Z 584.203,A -85,B 0,C 180,E1 -27212.16,E2 -27212.16} C_VEL
LIN {X 0,Y 127.764,Z 582.902,A -85,B 0,C 180,E1 -27213.373,E2 -27213.373} C_VEL
LIN {X 0,Y 127.594,Z 584.163,A -85,B 0,C 180,E1 -27214.282,E2 -27214.282} C_VEL
LIN {X 0,Y 119.842,Z 593.736,A -85,B 0,C 180,E1 -27217.65,E2 -27217.65} C_VEL
LIN {X 0,Y 112.689,Z 601.665,A -85,B 0,C 180,E1 -27221.542,E2 -27221.542} C_VEL
LIN {X 0,Y 105.978,Z 608.259,A -85,B 0,C 180,E1 -27225.862,E2 -27225.862} C_VEL
LIN {X 0,Y 99.961,Z 613.728,A -85,B 0,C 180,E1 -27230.739,E2 -27230.739} C_VEL
LIN {X 0,Y 93.43,Z 619.444,A -85,B 0,C 180,E1 -27238.221,E2 -27238.221} C_VEL
LIN {X 0,Y 88.286,Z 623.596,A -85,B 0,C 180,E1 -27246.539,E2 -27246.539} C_VEL
LIN {X 0,Y 85.141,Z 626.31,A -85,B 0,C 180,E1 -27255.656,E2 -27255.656} C_VEL
LIN {X 0,Y 83.805,Z 627.668,A -85,B 0,C 180,E1 -27265.183,E2 -27265.183} C_VEL
LIN {X 0,Y 83.813,Z 627.845,A -85,B 0,C 180,E1 -27269.994,E2 -27269.994} C_VEL
LIN {X 0,Y 84.23,Z 627.203,A -85,B 0,C 180,E1 -27279.6,E2 -27279.6} C_VEL
LIN {X 0,Y 86.451,Z 625.214,A -85,B 0,C 180,E1 -27288.97,E2 -27288.97} C_VEL
LIN {X 0,Y 90.541,Z 621.831,A -85,B 0,C 180,E1 -27297.751,E2 -27297.751} C_VEL
LIN {X 0,Y 94.894,Z 618.352,A -85,B 0,C 180,E1 -27303.736,E2 -27303.736} C_VEL
LIN {X 0,Y 101.661,Z 612.402,A -85,B 0,C 180,E1 -27310.783,E2 -27310.783} C_VEL
LIN {X 0,Y 109.183,Z 605.368,A -85,B 0,C 180,E1 -27316.391,E2 -27316.391} C_VEL
LIN {X 0,Y 117.338,Z 596.852,A -85,B 0,C 180,E1 -27321.129,E2 -27321.129} C_VEL
LIN {X 0,Y 124.945,Z 587.938,A -85,B 0,C 180,E1 -27324.64,E2 -27324.64} C_VEL
LIN {X 0,Y 129.558,Z 581.83,A -85,B 0,C 180,E1 -27326.581,E2 -27326.581} C_VEL
LIN {X 0,Y 132.626,Z 574.042,A -85,B 0,C 180,E1 -27330.187,E2 -27330.187} C_VEL
LIN {X 0,Y 133.559,Z 570.925,A -85,B 0,C 180,E1 -27331.732,E2 -27331.732} C_VEL
LIN {X 0,Y 133.755,Z 566.023,A -85,B 0,C 180,E1 -27335.143,E2 -27335.143} C_VEL
LIN {X 0,Y 133.619,Z 561.91,A -85,B 0,C 180,E1 -27338.396,E2 -27338.396} C_VEL
LIN {X 0,Y 133.143,Z 557.173,A -85,B 0,C 180,E1 -27342.965,E2 -27342.965} C_VEL
LIN {X 0,Y 132.666,Z 553.272,A -85,B 0,C 180,E1 -27347.766,E2 -27347.766} C_VEL
LIN {X 0,Y 132.441,Z 551.359,A -85,B 0,C 180,E1 -27350.84,E2 -27350.84} C_VEL
LIN {X 0,Y 132.242,Z 550.078,A -85,B 0,C 180,E1 -27353.898,E2 -27353.898} C_VEL
LIN {X 0,Y 132.395,Z 548.415,A -85,B 0,C 180,E1 -27360,E2 -27360} C_VEL
LIN {X 0,Y 132.485,Z 549.76,A -85,B 0,C 180,E1 -27366.09,E2 -27366.09} C_VEL
LIN {X 0,Y 132.788,Z 550.931,A -85,B 0,C 180,E1 -27369.136,E2 -27369.136} C_VEL
LIN {X 0,Y 133.456,Z 553.55,A -85,B 0,C 180,E1 -27373.708,E2 -27373.708} C_VEL
LIN {X 0,Y 134.356,Z 557.157,A -85,B 0,C 180,E1 -27378.291,E2 -27378.291} C_VEL
LIN {X 0,Y 134.949,Z 560.244,A -85,B 0,C 180,E1 -27381.38,E2 -27381.38} C_VEL
LIN {X 0,Y 135.605,Z 564.943,A -85,B 0,C 180,E1 -27385.353,E2 -27385.353} C_VEL
LIN {X 0,Y 135.729,Z 567.346,A -85,B 0,C 180,E1 -27387.043,E2 -27387.043} C_VEL
LIN {X 0,Y 135.402,Z 570.915,A -85,B 0,C 180,E1 -27389.187,E2 -27389.187} C_VEL
LIN {X 0,Y 135.085,Z 572.567,A -85,B 0,C 180,E1 -27390.023,E2 -27390.023} C_VEL
LIN {X 0,Y 132.422,Z 578.014,A -85,B 0,C 180,E1 -27391.887,E2 -27391.887} C_VEL
LIN {X 0,Y 125.87,Z 587.26,A -85,B 0,C 180,E1 -27394.564,E2 -27394.564} C_VEL
LIN {X 0,Y 118.165,Z 596.526,A -85,B 0,C 180,E1 -27398.003,E2 -27398.003} C_VEL
LIN {X 0,Y 110.993,Z 604.22,A -85,B 0,C 180,E1 -27401.934,E2 -27401.934} C_VEL
LIN {X 0,Y 103.389,Z 611.557,A -85,B 0,C 180,E1 -27407.182,E2 -27407.182} C_VEL
LIN {X 0,Y 97.442,Z 616.853,A -85,B 0,C 180,E1 -27412.502,E2 -27412.502} C_VEL
LIN {X 0,Y 91.504,Z 621.992,A -85,B 0,C 180,E1 -27420.057,E2 -27420.057} C_VEL
LIN {X 0,Y 87.869,Z 624.944,A -85,B 0,C 180,E1 -27426.434,E2 -27426.434} C_VEL
LIN {X 0,Y 84.906,Z 627.657,A -85,B 0,C 180,E1 -27435.628,E2 -27435.628} C_VEL
LIN {X 0,Y 83.761,Z 628.998,A -85,B 0,C 180,E1 -27445.193,E2 -27445.193} C_VEL
LIN {X 0,Y 83.809,Z 629.161,A -85,B 0,C 180,E1 -27450.006,E2 -27450.006} C_VEL
LIN {X 0,Y 84.122,Z 628.464,A -85,B 0,C 180,E1 -27459.625,E2 -27459.625} C_VEL
LIN {X 0,Y 86.151,Z 626.414,A -85,B 0,C 180,E1 -27469.051,E2 -27469.051} C_VEL
LIN {X 0,Y 90.202,Z 622.966,A -85,B 0,C 180,E1 -27477.877,E2 -27477.877} C_VEL
LIN {X 0,Y 96.194,Z 618.019,A -85,B 0,C 180,E1 -27485.773,E2 -27485.773} C_VEL
LIN {X 0,Y 101.845,Z 613.218,A -85,B 0,C 180,E1 -27490.969,E2 -27490.969} C_VEL
LIN {X 0,Y 109.794,Z 606.281,A -85,B 0,C 180,E1 -27496.071,E2 -27496.071} C_VEL
LIN {X 0,Y 111.019,Z 605.173,A -85,B 0,C 180,E1 -27496.725,E2 -27496.725} C_VEL
LIN {X 0,Y 111.296,Z 604.071,A -85,B 0,C 180,E1 -27497.86,E2 -27497.86} C_VEL
LIN {X 0,Y 98.049,Z 602.286,A -85,B 0,C 180,E1 -27509.885,E2 -27509.885} C_VEL
LIN {X 0,Y 93.832,Z 600.657,A -85,B 0,C 180,E1 -27518.007,E2 -27518.007} C_VEL
LIN {X 0,Y 92.091,Z 600.117,A -85,B 0,C 180,E1 -27522.226,E2 -27522.226} C_VEL
LIN {X 0,Y 91.376,Z 598.038,A -85,B 0,C 180,E1 -27531.152,E2 -27531.152} C_VEL
LIN {X 0,Y 91.612,Z 597.154,A -85,B 0,C 180,E1 -27535.853,E2 -27535.853} C_VEL
LIN {X 0,Y 92.727,Z 596.069,A -85,B 0,C 180,E1 -27540,E2 -27540} C_VEL
LIN {X 0,Y 104.523,Z 591.029,A -85,B 0,C 180,E1 -27559.646,E2 -27559.646} C_VEL
LIN {X 0,Y 117.277,Z 586.767,A -85,B 0,C 180,E1 -27568.647,E2 -27568.647} C_VEL
LIN {X 0,Y 119.763,Z 585.879,A -85,B 0,C 180,E1 -27569.929,E2 -27569.929} C_VEL
LIN {X 0,Y 120.544,Z 586.044,A -85,B 0,C 180,E1 -27570.721,E2 -27570.721} C_VEL
LIN {X 0,Y 120.444,Z 587.364,A -85,B 0,C 180,E1 -27571.934,E2 -27571.934} C_VEL
LIN {X 0,Y 119.282,Z 589.563,A -85,B 0,C 180,E1 -27573.187,E2 -27573.187} C_VEL
LIN {X 0,Y 114.945,Z 594.719,A -85,B 0,C 180,E1 -27575.335,E2 -27575.335} C_VEL
LIN {X 0,Y 111.009,Z 598.791,A -85,B 0,C 180,E1 -27577.14,E2 -27577.14} C_VEL
LIN {X 0,Y 103.286,Z 606.273,A -85,B 0,C 180,E1 -27581.534,E2 -27581.534} C_VEL
LIN {X 0,Y 96.625,Z 612.074,A -85,B 0,C 180,E1 -27586.286,E2 -27586.286} C_VEL
LIN {X 0,Y 89.092,Z 618.254,A -85,B 0,C 180,E1 -27593.72,E2 -27593.72} C_VEL
LIN {X 0,Y 84.374,Z 621.762,A -85,B 0,C 180,E1 -27600.008,E2 -27600.008} C_VEL
LIN {X 0,Y 79.765,Z 625.183,A -85,B 0,C 180,E1 -27609.357,E2 -27609.357} C_VEL
LIN {X 0,Y 77.24,Z 627.212,A -85,B 0,C 180,E1 -27619.508,E2 -27619.508} C_VEL
LIN {X 0,Y 76.734,Z 627.901,A -85,B 0,C 180,E1 -27629.993,E2 -27629.993} C_VEL
LIN {X 0,Y 77.235,Z 627.259,A -85,B 0,C 180,E1 -27640.479,E2 -27640.479} C_VEL
LIN {X 0,Y 79.734,Z 625.269,A -85,B 0,C 180,E1 -27650.638,E2 -27650.638} C_VEL
LIN {X 0,Y 84.314,Z 621.886,A -85,B 0,C 180,E1 -27660.001,E2 -27660.001} C_VEL
LIN {X 0,Y 90.781,Z 617.006,A -85,B 0,C 180,E1 -27668.26,E2 -27668.26} C_VEL
LIN {X 0,Y 98.69,Z 610.487,A -85,B 0,C 180,E1 -27675.401,E2 -27675.401} C_VEL
LIN {X 0,Y 106.787,Z 603.205,A -85,B 0,C 180,E1 -27680.643,E2 -27680.643} C_VEL
LIN {X 0,Y 115.589,Z 594.12,A -85,B 0,C 180,E1 -27685.159,E2 -27685.159} C_VEL
LIN {X 0,Y 123.681,Z 584.61,A -85,B 0,C 180,E1 -27688.46,E2 -27688.46} C_VEL
LIN {X 0,Y 124.788,Z 583.129,A -85,B 0,C 180,E1 -27688.934,E2 -27688.934} C_VEL
LIN {X 0,Y 128.107,Z 575.722,A -85,B 0,C 180,E1 -27692.576,E2 -27692.576} C_VEL
LIN {X 0,Y 128.634,Z 573.353,A -85,B 0,C 180,E1 -27694.082,E2 -27694.082} C_VEL
LIN {X 0,Y 128.998,Z 568.594,A -85,B 0,C 180,E1 -27697.836,E2 -27697.836} C_VEL
LIN {X 0,Y 128.975,Z 564.257,A -85,B 0,C 180,E1 -27701.978,E2 -27701.978} C_VEL
LIN {X 0,Y 128.917,Z 560.911,A -85,B 0,C 180,E1 -27705.799,E2 -27705.799} C_VEL
LIN {X 0,Y 128.72,Z 557.774,A -85,B 0,C 180,E1 -27710.572,E2 -27710.572} C_VEL
LIN {X 0,Y 128.663,Z 556.353,A -85,B 0,C 180,E1 -27713.728,E2 -27713.728} C_VEL
LIN {X 0,Y 128.944,Z 554.659,A -85,B 0,C 180,E1 -27720,E2 -27720} C_VEL
LIN {X 0,Y 128.868,Z 555.166,A -85,B 0,C 180,E1 -27723.126,E2 -27723.126} C_VEL
LIN {X 0,Y 128.943,Z 556.043,A -85,B 0,C 180,E1 -27726.258,E2 -27726.258} C_VEL
LIN {X 0,Y 129.158,Z 557.278,A -85,B 0,C 180,E1 -27729.395,E2 -27729.395} C_VEL
LIN {X 0,Y 129.683,Z 559.985,A -85,B 0,C 180,E1 -27734.115,E2 -27734.115} C_VEL
LIN {X 0,Y 130.294,Z 563.785,A -85,B 0,C 180,E1 -27738.883,E2 -27738.883} C_VEL
LIN {X 0,Y 130.696,Z 568.131,A -85,B 0,C 180,E1 -27743.059,E2 -27743.059} C_VEL
LIN {X 0,Y 130.789,Z 571.019,A -85,B 0,C 180,E1 -27745.46,E2 -27745.46} C_VEL
LIN {X 0,Y 130.287,Z 574.486,A -85,B 0,C 180,E1 -27747.713,E2 -27747.713} C_VEL
LIN {X 0,Y 128.641,Z 577.968,A -85,B 0,C 180,E1 -27749.068,E2 -27749.068} C_VEL
LIN {X 0,Y 127.181,Z 580.285,A -85,B 0,C 180,E1 -27749.824,E2 -27749.824} C_VEL
LIN {X 0,Y 119.275,Z 590.465,A -85,B 0,C 180,E1 -27752.906,E2 -27752.906} C_VEL
LIN {X 0,Y 111.303,Z 599.169,A -85,B 0,C 180,E1 -27756.391,E2 -27756.391} C_VEL
LIN {X 0,Y 102.789,Z 607.508,A -85,B 0,C 180,E1 -27761.235,E2 -27761.235} C_VEL
LIN {X 0,Y 96.129,Z 613.304,A -85,B 0,C 180,E1 -27766.017,E2 -27766.017} C_VEL
LIN {X 0,Y 90.264,Z 618.074,A -85,B 0,C 180,E1 -27771.481,E2 -27771.481} C_VEL
LIN {X 0,Y 83.954,Z 622.999,A -85,B 0,C 180,E1 -27779.857,E2 -27779.857} C_VEL
LIN {X 0,Y 79.432,Z 626.42,A -85,B 0,C 180,E1 -27789.28,E2 -27789.28} C_VEL
LIN {X 0,Y 77.106,Z 628.442,A -85,B 0,C 180,E1 -27799.503,E2 -27799.503} C_VEL
LIN {X 0,Y 76.707,Z 629.105,A -85,B 0,C 180,E1 -27810.007,E2 -27810.007} C_VEL
LIN {X 0,Y 77.109,Z 628.408,A -85,B 0,C 180,E1 -27820.51,E2 -27820.51} C_VEL
LIN {X 0,Y 79.436,Z 626.358,A -85,B 0,C 180,E1 -27830.732,E2 -27830.732} C_VEL
LIN {X 0,Y 83.967,Z 622.91,A -85,B 0,C 180,E1 -27840.152,E2 -27840.152} C_VEL
LIN {X 0,Y 90.498,Z 617.962,A -85,B 0,C 180,E1 -27848.416,E2 -27848.416} C_VEL
LIN {X 0,Y 96.595,Z 613.162,A -85,B 0,C 180,E1 -27853.732,E2 -27853.732} C_VEL
LIN {X 0,Y 102.628,Z 608.243,A -85,B 0,C 180,E1 -27857.617,E2 -27857.617} C_VEL
LIN {X 0,Y 102.025,Z 607.422,A -85,B 0,C 180,E1 -27859.128,E2 -27859.128} C_VEL
LIN {X 0,Y 92.94,Z 606.213,A -85,B 0,C 180,E1 -27868.04,E2 -27868.04} C_VEL
LIN {X 0,Y 88.328,Z 604.728,A -85,B 0,C 180,E1 -27876.557,E2 -27876.557} C_VEL
LIN {X 0,Y 86.507,Z 604.186,A -85,B 0,C 180,E1 -27881.037,E2 -27881.037} C_VEL
LIN {X 0,Y 99.266,Z 595.718,A -85,B 0,C 180,E1 -27920.732,E2 -27920.732} C_VEL
LIN {X 0,Y 112.461,Z 591.762,A -85,B 0,C 180,E1 -27929.997,E2 -27929.997} C_VEL
LIN {X 0,Y 118.839,Z 589.751,A -85,B 0,C 180,E1 -27933.064,E2 -27933.064} C_VEL
LIN {X 0,Y 118.281,Z 590.837,A -85,B 0,C 180,E1 -27933.704,E2 -27933.704} C_VEL
LIN {X 0,Y 111.009,Z 598.791,A -85,B 0,C 180,E1 -27937.14,E2 -27937.14} C_VEL
LIN {X 0,Y 107.172,Z 602.253,A -85,B 0,C 180,E1 -27938.659,E2 -27938.659} C_VEL
LIN {X 0,Y 99.588,Z 607.466,A -85,B 0,C 180,E1 -27940.755,E2 -27940.755} C_VEL
LIN {X 0,Y 92.014,Z 612.105,A -85,B 0,C 180,E1 -27943.401,E2 -27943.401} C_VEL
LIN {X 0,Y 88.325,Z 614.624,A -85,B 0,C 180,E1 -27945.841,E2 -27945.841} C_VEL
LIN {X 0,Y 81.647,Z 619.556,A -85,B 0,C 180,E1 -27952.94,E2 -27952.94} C_VEL
LIN {X 0,Y 75.404,Z 623.708,A -85,B 0,C 180,E1 -27962.216,E2 -27962.216} C_VEL
LIN {X 0,Y 71.434,Z 626.423,A -85,B 0,C 180,E1 -27972.826,E2 -27972.826} C_VEL
LIN {X 0,Y 69.663,Z 627.779,A -85,B 0,C 180,E1 -27984.203,E2 -27984.203} C_VEL
LIN {X 0,Y 69.646,Z 627.956,A -85,B 0,C 180,E1 -27989.993,E2 -27989.993} C_VEL
LIN {X 0,Y 70.246,Z 627.314,A -85,B 0,C 180,E1 -28001.535,E2 -28001.535} C_VEL
LIN {X 0,Y 73.106,Z 625.324,A -85,B 0,C 180,E1 -28012.607,E2 -28012.607} C_VEL
LIN {X 0,Y 78.238,Z 621.94,A -85,B 0,C 180,E1 -28022.606,E2 -28022.606} C_VEL
LIN {X 0,Y 85.3,Z 617.06,A -85,B 0,C 180,E1 -28031.225,E2 -28031.225} C_VEL
LIN {X 0,Y 93.813,Z 610.539,A -85,B 0,C 180,E1 -28038.508,E2 -28038.508} C_VEL
LIN {X 0,Y 102.414,Z 603.256,A -85,B 0,C 180,E1 -28043.729,E2 -28043.729} C_VEL
LIN {X 0,Y 111.681,Z 594.169,A -85,B 0,C 180,E1 -28048.153,E2 -28048.153} C_VEL
LIN {X 0,Y 120.093,Z 584.657,A -85,B 0,C 180,E1 -28051.371,E2 -28051.371} C_VEL
LIN {X 0,Y 123.144,Z 578.699,A -85,B 0,C 180,E1 -28054.465,E2 -28054.465} C_VEL
LIN {X 0,Y 123.814,Z 575.888,A -85,B 0,C 180,E1 -28056.588,E2 -28056.588} C_VEL
LIN {X 0,Y 124.351,Z 571.885,A -85,B 0,C 180,E1 -28060.177,E2 -28060.177} C_VEL
LIN {X 0,Y 124.598,Z 567.308,A -85,B 0,C 180,E1 -28065.294,E2 -28065.294} C_VEL
LIN {X 0,Y 124.708,Z 563.976,A -85,B 0,C 180,E1 -28070.266,E2 -28070.266} C_VEL
LIN {X 0,Y 124.764,Z 562.481,A -85,B 0,C 180,E1 -28073.531,E2 -28073.531} C_VEL
LIN {X 0,Y 125.201,Z 560.727,A -85,B 0,C 180,E1 -28080,E2 -28080} C_VEL
LIN {X 0,Y 125.091,Z 561.244,A -85,B 0,C 180,E1 -28083.22,E2 -28083.22} C_VEL
LIN {X 0,Y 125.095,Z 562.151,A -85,B 0,C 180,E1 -28086.451,E2 -28086.451} C_VEL
LIN {X 0,Y 125.229,Z 563.44,A -85,B 0,C 180,E1 -28089.692,E2 -28089.692} C_VEL
LIN {X 0,Y 125.567,Z 566.284,A -85,B 0,C 180,E1 -28094.588,E2 -28094.588} C_VEL
LIN {X 0,Y 125.783,Z 569.103,A -85,B 0,C 180,E1 -28098.235,E2 -28098.235} C_VEL
LIN {X 0,Y 125.856,Z 573.813,A -85,B 0,C 180,E1 -28103.01,E2 -28103.01} C_VEL
LIN {X 0,Y 125.539,Z 576.398,A -85,B 0,C 180,E1 -28105.066,E2 -28105.066} C_VEL
LIN {X 0,Y 125.127,Z 577.921,A -85,B 0,C 180,E1 -28106.027,E2 -28106.027} C_VEL
LIN {X 0,Y 123.198,Z 581.028,A -85,B 0,C 180,E1 -28107.153,E2 -28107.153} C_VEL
LIN {X 0,Y 115.567,Z 590.417,A -85,B 0,C 180,E1 -28109.945,E2 -28109.945} C_VEL
LIN {X 0,Y 107.232,Z 599.119,A -85,B 0,C 180,E1 -28113.327,E2 -28113.327} C_VEL
LIN {X 0,Y 98.233,Z 607.456,A -85,B 0,C 180,E1 -28118.104,E2 -28118.104} C_VEL
LIN {X 0,Y 91.129,Z 613.251,A -85,B 0,C 180,E1 -28122.9,E2 -28122.9} C_VEL
LIN {X 0,Y 84.769,Z 618.02,A -85,B 0,C 180,E1 -28128.46,E2 -28128.46} C_VEL
LIN {X 0,Y 77.868,Z 622.944,A -85,B 0,C 180,E1 -28137.22,E2 -28137.22} C_VEL
LIN {X 0,Y 72.784,Z 626.365,A -85,B 0,C 180,E1 -28147.287,E2 -28147.287} C_VEL
LIN {X 0,Y 70.103,Z 628.386,A -85,B 0,C 180,E1 -28158.441,E2 -28158.441} C_VEL
LIN {X 0,Y 69.599,Z 629.049,A -85,B 0,C 180,E1 -28170.007,E2 -28170.007} C_VEL
LIN {X 0,Y 70.106,Z 628.352,A -85,B 0,C 180,E1 -28181.573,E2 -28181.573} C_VEL
LIN {X 0,Y 72.788,Z 626.301,A -85,B 0,C 180,E1 -28192.727,E2 -28192.727} C_VEL
LIN {X 0,Y 77.888,Z 622.854,A -85,B 0,C 180,E1 -28202.786,E2 -28202.786} C_VEL
LIN {X 0,Y 85.021,Z 617.907,A -85,B 0,C 180,E1 -28211.406,E2 -28211.406} C_VEL
LIN {X 0,Y 91.598,Z 613.107,A -85,B 0,C 180,E1 -28216.802,E2 -28216.802} C_VEL
LIN {X 0,Y 94.002,Z 611.308,A -85,B 0,C 180,E1 -28218.394,E2 -28218.394} C_VEL
LIN {X 0,Y 91.378,Z 610.29,A -85,B 0,C 180,E1 -28222.027,E2 -28222.027} C_VEL
LIN {X 0,Y 84.909,Z 609.234,A -85,B 0,C 180,E1 -28230.223,E2 -28230.223} C_VEL
LIN {X 0,Y 79.556,Z 606.946,A -85,B 0,C 180,E1 -28246.372,E2 -28246.372} C_VEL
LIN {X 0,Y 93.857,Z 600.103,A -85,B 0,C 180,E1 -28281.988,E2 -28281.988} C_VEL
LIN {X 0,Y 107.521,Z 596.467,A -85,B 0,C 180,E1 -28291.528,E2 -28291.528} C_VEL
LIN {X 0,Y 109.007,Z 596.654,A -85,B 0,C 180,E1 -28293.047,E2 -28293.047} C_VEL
LIN {X 0,Y 99.97,Z 605.223,A -85,B 0,C 180,E1 -28297.724,E2 -28297.724} C_VEL
LIN {X 0,Y 91.599,Z 612.13,A -85,B 0,C 180,E1 -28303.199,E2 -28303.199} C_VEL
LIN {X 0,Y 88.325,Z 614.624,A -85,B 0,C 180,E1 -28305.841,E2 -28305.841} C_VEL
LIN {X 0,Y 84.753,Z 616.977,A -85,B 0,C 180,E1 -28308.55,E2 -28308.55} C_VEL
LIN {X 0,Y 77.605,Z 620.38,A -85,B 0,C 180,E1 -28312.796,E2 -28312.796} C_VEL
LIN {X 0,Y 70.759,Z 623.176,A -85,B 0,C 180,E1 -28317.966,E2 -28317.966} C_VEL
LIN {X 0,Y 67.862,Z 624.502,A -85,B 0,C 180,E1 -28322.093,E2 -28322.093} C_VEL
LIN {X 0,Y 64.651,Z 626.479,A -85,B 0,C 180,E1 -28330.958,E2 -28330.958} C_VEL
LIN {X 0,Y 62.594,Z 627.835,A -85,B 0,C 180,E1 -28343.545,E2 -28343.545} C_VEL
LIN {X 0,Y 62.547,Z 628.012,A -85,B 0,C 180,E1 -28349.992,E2 -28349.992} C_VEL
LIN {X 0,Y 63.299,Z 627.37,A -85,B 0,C 180,E1 -28362.821,E2 -28362.821} C_VEL
LIN {X 0,Y 66.587,Z 625.379,A -85,B 0,C 180,E1 -28374.964,E2 -28374.964} C_VEL
LIN {X 0,Y 72.326,Z 621.995,A -85,B 0,C 180,E1 -28385.655,E2 -28385.655} C_VEL
LIN {X 0,Y 80.071,Z 617.113,A -85,B 0,C 180,E1 -28394.592,E2 -28394.592} C_VEL
LIN {X 0,Y 89.256,Z 610.592,A -85,B 0,C 180,E1 -28401.933,E2 -28401.933} C_VEL
LIN {X 0,Y 98.366,Z 603.307,A -85,B 0,C 180,E1 -28407.077,E2 -28407.077} C_VEL
LIN {X 0,Y 106.669,Z 595.661,A -85,B 0,C 180,E1 -28410.798,E2 -28410.798} C_VEL
LIN {X 0,Y 114.955,Z 586.947,A -85,B 0,C 180,E1 -28413.788,E2 -28413.788} C_VEL
LIN {X 0,Y 115.886,Z 585.743,A -85,B 0,C 180,E1 -28414.243,E2 -28414.243} C_VEL
LIN {X 0,Y 118.106,Z 581.961,A -85,B 0,C 180,E1 -28416.317,E2 -28416.317} C_VEL
LIN {X 0,Y 118.811,Z 579.549,A -85,B 0,C 180,E1 -28418.302,E2 -28418.302} C_VEL
LIN {X 0,Y 119.453,Z 576.668,A -85,B 0,C 180,E1 -28421.118,E2 -28421.118} C_VEL
LIN {X 0,Y 120.108,Z 572.229,A -85,B 0,C 180,E1 -28426.464,E2 -28426.464} C_VEL
LIN {X 0,Y 120.376,Z 570.007,A -85,B 0,C 180,E1 -28429.912,E2 -28429.912} C_VEL
LIN {X 0,Y 120.553,Z 568.445,A -85,B 0,C 180,E1 -28433.304,E2 -28433.304} C_VEL
LIN {X 0,Y 121.153,Z 566.634,A -85,B 0,C 180,E1 -28440,E2 -28440} C_VEL
LIN {X 0,Y 121.024,Z 567.129,A -85,B 0,C 180,E1 -28443.329,E2 -28443.329} C_VEL
LIN {X 0,Y 120.99,Z 568.987,A -85,B 0,C 180,E1 -28449.104,E2 -28449.104} C_VEL
LIN {X 0,Y 121.126,Z 572.398,A -85,B 0,C 180,E1 -28455.135,E2 -28455.135} C_VEL
LIN {X 0,Y 120.96,Z 576.745,A -85,B 0,C 180,E1 -28460.402,E2 -28460.402} C_VEL
LIN {X 0,Y 120.548,Z 579.652,A -85,B 0,C 180,E1 -28463.173,E2 -28463.173} C_VEL
LIN {X 0,Y 120.187,Z 580.737,A -85,B 0,C 180,E1 -28463.946,E2 -28463.946} C_VEL
LIN {X 0,Y 116.559,Z 585.355,A -85,B 0,C 180,E1 -28465.264,E2 -28465.264} C_VEL
LIN {X 0,Y 107.798,Z 594.923,A -85,B 0,C 180,E1 -28468.351,E2 -28468.351} C_VEL
LIN {X 0,Y 99.328,Z 602.849,A -85,B 0,C 180,E1 -28471.9,E2 -28471.9} C_VEL
LIN {X 0,Y 91.394,Z 609.437,A -85,B 0,C 180,E1 -28476.165,E2 -28476.165} C_VEL
LIN {X 0,Y 84.046,Z 614.9,A -85,B 0,C 180,E1 -28481.195,E2 -28481.195} C_VEL
LIN {X 0,Y 75.556,Z 620.624,A -85,B 0,C 180,E1 -28489.384,E2 -28489.384} C_VEL
LIN {X 0,Y 68.786,Z 624.78,A -85,B 0,C 180,E1 -28499.288,E2 -28499.288} C_VEL
LIN {X 0,Y 64.405,Z 627.491,A -85,B 0,C 180,E1 -28510.9,E2 -28510.9} C_VEL
LIN {X 0,Y 62.528,Z 628.831,A -85,B 0,C 180,E1 -28523.555,E2 -28523.555} C_VEL
LIN {X 0,Y 62.51,Z 628.994,A -85,B 0,C 180,E1 -28530.008,E2 -28530.008} C_VEL
LIN {X 0,Y 63.146,Z 628.296,A -85,B 0,C 180,E1 -28542.87,E2 -28542.87} C_VEL
LIN {X 0,Y 66.248,Z 626.245,A -85,B 0,C 180,E1 -28555.117,E2 -28555.117} C_VEL
LIN {X 0,Y 72.001,Z 622.798,A -85,B 0,C 180,E1 -28565.858,E2 -28565.858} C_VEL
LIN {X 0,Y 79.802,Z 617.851,A -85,B 0,C 180,E1 -28574.801,E2 -28574.801} C_VEL
LIN {X 0,Y 84.415,Z 614.769,A -85,B 0,C 180,E1 -28578.538,E2 -28578.538} C_VEL
LIN {X 0,Y 85.35,Z 613.48,A -85,B 0,C 180,E1 -28580.561,E2 -28580.561} C_VEL
LIN {X 0,Y 79.49,Z 612.635,A -85,B 0,C 180,E1 -28587.962,E2 -28587.962} C_VEL
LIN {X 0,Y 73.716,Z 610.804,A -85,B 0,C 180,E1 -28603.381,E2 -28603.381} C_VEL
LIN {X 0,Y 88.299,Z 604.208,A -85,B 0,C 180,E1 -28643.451,E2 -28643.451} C_VEL
LIN {X 0,Y 98.36,Z 601.85,A -85,B 0,C 180,E1 -28650.963,E2 -28650.963} C_VEL
LIN {X 0,Y 99.788,Z 601.829,A -85,B 0,C 180,E1 -28652.303,E2 -28652.303} C_VEL
LIN {X 0,Y 91.846,Z 608.424,A -85,B 0,C 180,E1 -28656.53,E2 -28656.53} C_VEL
LIN {X 0,Y 82.715,Z 615.13,A -85,B 0,C 180,E1 -28662.952,E2 -28662.952} C_VEL
LIN {X 0,Y 76.057,Z 619.612,A -85,B 0,C 180,E1 -28669.688,E2 -28669.688} C_VEL
LIN {X 0,Y 69.172,Z 623.764,A -85,B 0,C 180,E1 -28679.46,E2 -28679.46} C_VEL
LIN {X 0,Y 67.862,Z 624.502,A -85,B 0,C 180,E1 -28682.093,E2 -28682.093} C_VEL
LIN {X 0,Y 65.322,Z 625.714,A -85,B 0,C 180,E1 -28686.572,E2 -28686.572} C_VEL
LIN {X 0,Y 60.208,Z 627.094,A -85,B 0,C 180,E1 -28694.233,E2 -28694.233} C_VEL
LIN {X 0,Y 56.744,Z 627.776,A -85,B 0,C 180,E1 -28701.259,E2 -28701.259} C_VEL
LIN {X 0,Y 55.471,Z 628.01,A -85,B 0,C 180,E1 -28707.187,E2 -28707.187} C_VEL
LIN {X 0,Y 55.433,Z 628.049,A -85,B 0,C 180,E1 -28709.233,E2 -28709.233} C_VEL
LIN {X 0,Y 55.548,Z 627.914,A -85,B 0,C 180,E1 -28717.259,E2 -28717.259} C_VEL
LIN {X 0,Y 57.946,Z 626.599,A -85,B 0,C 180,E1 -28731.327,E2 -28731.327} C_VEL
LIN {X 0,Y 63.071,Z 623.922,A -85,B 0,C 180,E1 -28743.849,E2 -28743.849} C_VEL
LIN {X 0,Y 70.69,Z 619.803,A -85,B 0,C 180,E1 -28754.092,E2 -28754.092} C_VEL
LIN {X 0,Y 79.922,Z 614.122,A -85,B 0,C 180,E1 -28762.307,E2 -28762.307} C_VEL
LIN {X 0,Y 89.103,Z 607.7,A -85,B 0,C 180,E1 -28767.973,E2 -28767.973} C_VEL
LIN {X 0,Y 98.998,Z 599.71,A -85,B 0,C 180,E1 -28772.535,E2 -28772.535} C_VEL
LIN {X 0,Y 107.884,Z 591.326,A -85,B 0,C 180,E1 -28775.773,E2 -28775.773} C_VEL
LIN {X 0,Y 111.708,Z 587.192,A -85,B 0,C 180,E1 -28777.122,E2 -28777.122} C_VEL
LIN {X 0,Y 113.252,Z 584.762,A -85,B 0,C 180,E1 -28778.554,E2 -28778.554} C_VEL
LIN {X 0,Y 114.428,Z 581.244,A -85,B 0,C 180,E1 -28782.116,E2 -28782.116} C_VEL
LIN {X 0,Y 115.344,Z 577.418,A -85,B 0,C 180,E1 -28787.111,E2 -28787.111} C_VEL
LIN {X 0,Y 115.712,Z 575.875,A -85,B 0,C 180,E1 -28789.501,E2 -28789.501} C_VEL
LIN {X 0,Y 116.032,Z 574.231,A -85,B 0,C 180,E1 -28793.042,E2 -28793.042} C_VEL
LIN {X 0,Y 116.364,Z 573.102,A -85,B 0,C 180,E1 -28796.537,E2 -28796.537} C_VEL
LIN {X 0,Y 116.817,Z 572.342,A -85,B 0,C 180,E1 -28800,E2 -28800} C_VEL
LIN {X 0,Y 116.654,Z 572.837,A -85,B 0,C 180,E1 -28803.454,E2 -28803.454} C_VEL
LIN {X 0,Y 116.515,Z 573.816,A -85,B 0,C 180,E1 -28806.929,E2 -28806.929} C_VEL
LIN {X 0,Y 116.398,Z 575.293,A -85,B 0,C 180,E1 -28810.436,E2 -28810.436} C_VEL
LIN {X 0,Y 116.334,Z 577.765,A -85,B 0,C 180,E1 -28814.87,E2 -28814.87} C_VEL
LIN {X 0,Y 115.88,Z 581.332,A -85,B 0,C 180,E1 -28819.485,E2 -28819.485} C_VEL
LIN {X 0,Y 115.494,Z 583.186,A -85,B 0,C 180,E1 -28821.414,E2 -28821.414} C_VEL
LIN {X 0,Y 107.626,Z 591.922,A -85,B 0,C 180,E1 -28823.92,E2 -28823.92} C_VEL
LIN {X 0,Y 98.651,Z 600.348,A -85,B 0,C 180,E1 -28827.074,E2 -28827.074} C_VEL
LIN {X 0,Y 88.744,Z 608.383,A -85,B 0,C 180,E1 -28831.654,E2 -28831.654} C_VEL
LIN {X 0,Y 79.517,Z 614.846,A -85,B 0,C 180,E1 -28837.313,E2 -28837.313} C_VEL
LIN {X 0,Y 70.287,Z 620.57,A -85,B 0,C 180,E1 -28845.589,E2 -28845.589} C_VEL
LIN {X 0,Y 62.768,Z 624.725,A -85,B 0,C 180,E1 -28855.965,E2 -28855.965} C_VEL
LIN {X 0,Y 57.693,Z 627.435,A -85,B 0,C 180,E1 -28868.574,E2 -28868.574} C_VEL
LIN {X 0,Y 55.467,Z 628.776,A -85,B 0,C 180,E1 -28882.73,E2 -28882.73} C_VEL
LIN {X 0,Y 55.407,Z 628.938,A -85,B 0,C 180,E1 -28890.009,E2 -28890.009} C_VEL
LIN {X 0,Y 56.238,Z 628.24,A -85,B 0,C 180,E1 -28904.483,E2 -28904.483} C_VEL
LIN {X 0,Y 59.852,Z 626.189,A -85,B 0,C 180,E1 -28918.024,E2 -28918.024} C_VEL
LIN {X 0,Y 66.342,Z 622.742,A -85,B 0,C 180,E1 -28929.475,E2 -28929.475} C_VEL
LIN {X 0,Y 74.908,Z 617.795,A -85,B 0,C 180,E1 -28938.65,E2 -28938.65} C_VEL
LIN {X 0,Y 76.584,Z 616.793,A -85,B 0,C 180,E1 -28940.031,E2 -28940.031} C_VEL
LIN {X 0,Y 74.089,Z 615.729,A -85,B 0,C 180,E1 -28945.309,E2 -28945.309} C_VEL
LIN {X 0,Y 67.581,Z 614.065,A -85,B 0,C 180,E1 -28961.822,E2 -28961.822} C_VEL
LIN {X 0,Y 87.156,Z 607.114,A -85,B 0,C 180,E1 -29008.936,E2 -29008.936} C_VEL
LIN {X 0,Y 90.556,Z 606.437,A -85,B 0,C 180,E1 -29011.374,E2 -29011.374} C_VEL
LIN {X 0,Y 82.491,Z 612.241,A -85,B 0,C 180,E1 -29015.956,E2 -29015.956} C_VEL
LIN {X 0,Y 75.173,Z 617.015,A -85,B 0,C 180,E1 -29021.579,E2 -29021.579} C_VEL
LIN {X 0,Y 66.735,Z 621.931,A -85,B 0,C 180,E1 -29030.802,E2 -29030.802} C_VEL
LIN {X 0,Y 60.228,Z 625.351,A -85,B 0,C 180,E1 -29042.167,E2 -29042.167} C_VEL
LIN {X 0,Y 56.384,Z 627.38,A -85,B 0,C 180,E1 -29055.555,E2 -29055.555} C_VEL
LIN {X 0,Y 55.433,Z 628.049,A -85,B 0,C 180,E1 -29069.233,E2 -29069.233} C_VEL
LIN {X 0,Y 55.299,Z 628.091,A -85,B 0,C 180,E1 -29073.283,E2 -29073.283} C_VEL
LIN {X 0,Y 54.765,Z 628.024,A -85,B 0,C 180,E1 -29077.336,E2 -29077.336} C_VEL
LIN {X 0,Y 53.332,Z 627.57,A -85,B 0,C 180,E1 -29085.617,E2 -29085.617} C_VEL
LIN {X 0,Y 52.717,Z 626.656,A -85,B 0,C 180,E1 -29094.264,E2 -29094.264} C_VEL
LIN {X 0,Y 53.741,Z 625.651,A -85,B 0,C 180,E1 -29100.538,E2 -29100.538} C_VEL
LIN {X 0,Y 54.476,Z 625.245,A -85,B 0,C 180,E1 -29102.461,E2 -29102.461} C_VEL
LIN {X 0,Y 61.306,Z 622.104,A -85,B 0,C 180,E1 -29113.447,E2 -29113.447} C_VEL
LIN {X 0,Y 70.615,Z 617.221,A -85,B 0,C 180,E1 -29122.757,E2 -29122.757} C_VEL
LIN {X 0,Y 81.244,Z 610.697,A -85,B 0,C 180,E1 -29129.875,E2 -29129.875} C_VEL
LIN {X 0,Y 91.407,Z 603.409,A -85,B 0,C 180,E1 -29134.597,E2 -29134.597} C_VEL
LIN {X 0,Y 100.489,Z 595.76,A -85,B 0,C 180,E1 -29137.908,E2 -29137.908} C_VEL
LIN {X 0,Y 107.189,Z 589.318,A -85,B 0,C 180,E1 -29139.88,E2 -29139.88} C_VEL
LIN {X 0,Y 108.477,Z 587.516,A -85,B 0,C 180,E1 -29141.098,E2 -29141.098} C_VEL
LIN {X 0,Y 109.501,Z 584.839,A -85,B 0,C 180,E1 -29144.29,E2 -29144.29} C_VEL
LIN {X 0,Y 110.633,Z 581.655,A -85,B 0,C 180,E1 -29149.013,E2 -29149.013} C_VEL
LIN {X 0,Y 111.203,Z 579.827,A -85,B 0,C 180,E1 -29152.738,E2 -29152.738} C_VEL
LIN {X 0,Y 111.667,Z 578.625,A -85,B 0,C 180,E1 -29156.391,E2 -29156.391} C_VEL
LIN {X 0,Y 112.212,Z 577.827,A -85,B 0,C 180,E1 -29160,E2 -29160} C_VEL
LIN {X 0,Y 112.008,Z 578.338,A -85,B 0,C 180,E1 -29163.597,E2 -29163.597} C_VEL
LIN {X 0,Y 111.763,Z 579.384,A -85,B 0,C 180,E1 -29167.225,E2 -29167.225} C_VEL
LIN {X 0,Y 111.463,Z 581.824,A -85,B 0,C 180,E1 -29172.749,E2 -29172.749} C_VEL
LIN {X 0,Y 110.988,Z 584.257,A -85,B 0,C 180,E1 -29176.557,E2 -29176.557} C_VEL
LIN {X 0,Y 110.626,Z 585.776,A -85,B 0,C 180,E1 -29178.52,E2 -29178.52} C_VEL
LIN {X 0,Y 110.029,Z 586.594,A -85,B 0,C 180,E1 -29178.92,E2 -29178.92} C_VEL
LIN {X 0,Y 100.259,Z 596.28,A -85,B 0,C 180,E1 -29181.766,E2 -29181.766} C_VEL
LIN {X 0,Y 91.094,Z 603.965,A -85,B 0,C 180,E1 -29184.985,E2 -29184.985} C_VEL
LIN {X 0,Y 80.918,Z 611.293,A -85,B 0,C 180,E1 -29189.725,E2 -29189.725} C_VEL
LIN {X 0,Y 70.183,Z 617.859,A -85,B 0,C 180,E1 -29196.777,E2 -29196.777} C_VEL
LIN {X 0,Y 60.945,Z 622.78,A -85,B 0,C 180,E1 -29206.231,E2 -29206.231} C_VEL
LIN {X 0,Y 53.642,Z 626.199,A -85,B 0,C 180,E1 -29218.406,E2 -29218.406} C_VEL
LIN {X 0,Y 49.357,Z 628.22,A -85,B 0,C 180,E1 -29233.465,E2 -29233.465} C_VEL
LIN {X 0,Y 48.32,Z 628.882,A -85,B 0,C 180,E1 -29250.011,E2 -29250.011} C_VEL
LIN {X 0,Y 49.361,Z 628.184,A -85,B 0,C 180,E1 -29266.555,E2 -29266.555} C_VEL
LIN {X 0,Y 53.649,Z 626.132,A -85,B 0,C 180,E1 -29281.612,E2 -29281.612} C_VEL
LIN {X 0,Y 60.986,Z 622.685,A -85,B 0,C 180,E1 -29293.755,E2 -29293.755} C_VEL
LIN {X 0,Y 65.494,Z 620.408,A -85,B 0,C 180,E1 -29298.701,E2 -29298.701} C_VEL
LIN {X 0,Y 68.5,Z 618.642,A -85,B 0,C 180,E1 -29302.006,E2 -29302.006} C_VEL
LIN {X 0,Y 63.666,Z 617.641,A -85,B 0,C 180,E1 -29312.036,E2 -29312.036} C_VEL
LIN {X 0,Y 60.727,Z 615.727,A -85,B 0,C 180,E1 -29333.355,E2 -29333.355} C_VEL
LIN {X 0,Y 80.081,Z 610.953,A -85,B 0,C 180,E1 -29369.895,E2 -29369.895} C_VEL
LIN {X 0,Y 78.062,Z 612.595,A -85,B 0,C 180,E1 -29372.018,E2 -29372.018} C_VEL
LIN {X 0,Y 70.633,Z 617.071,A -85,B 0,C 180,E1 -29377.239,E2 -29377.239} C_VEL
LIN {X 0,Y 61.372,Z 621.987,A -85,B 0,C 180,E1 -29386.589,E2 -29386.589} C_VEL
LIN {X 0,Y 54.029,Z 625.408,A -85,B 0,C 180,E1 -29398.636,E2 -29398.636} C_VEL
LIN {X 0,Y 49.53,Z 627.436,A -85,B 0,C 180,E1 -29413.503,E2 -29413.503} C_VEL
LIN {X 0,Y 48.367,Z 628.123,A -85,B 0,C 180,E1 -29429.989,E2 -29429.989} C_VEL
LIN {X 0,Y 49.523,Z 627.481,A -85,B 0,C 180,E1 -29446.478,E2 -29446.478} C_VEL
LIN {X 0,Y 53.992,Z 625.489,A -85,B 0,C 180,E1 -29461.366,E2 -29461.366} C_VEL
LIN {X 0,Y 54.476,Z 625.245,A -85,B 0,C 180,E1 -29462.461,E2 -29462.461} C_VEL
LIN {X 0,Y 56.627,Z 624.053,A -85,B 0,C 180,E1 -29467.989,E2 -29467.989} C_VEL
LIN {X 0,Y 59.703,Z 621.68,A -85,B 0,C 180,E1 -29476.998,E2 -29476.998} C_VEL
LIN {X 0,Y 62.92,Z 619.423,A -85,B 0,C 180,E1 -29483.471,E2 -29483.471} C_VEL
LIN {X 0,Y 66.306,Z 617.419,A -85,B 0,C 180,E1 -29487.405,E2 -29487.405} C_VEL
LIN {X 0,Y 67.662,Z 616.68,A -85,B 0,C 180,E1 -29488.466,E2 -29488.466} C_VEL
LIN {X 0,Y 77.917,Z 610.749,A -85,B 0,C 180,E1 -29494.404,E2 -29494.404} C_VEL
LIN {X 0,Y 88.583,Z 603.46,A -85,B 0,C 180,E1 -29498.767,E2 -29498.767} C_VEL
LIN {X 0,Y 98.033,Z 595.809,A -85,B 0,C 180,E1 -29501.767,E2 -29501.767} C_VEL
LIN {X 0,Y 102.868,Z 591.422,A -85,B 0,C 180,E1 -29503.017,E2 -29503.017} C_VEL
LIN {X 0,Y 103.904,Z 589.944,A -85,B 0,C 180,E1 -29504.302,E2 -29504.302} C_VEL
LIN {X 0,Y 105.193,Z 587.214,A -85,B 0,C 180,E1 -29508.437,E2 -29508.437} C_VEL
LIN {X 0,Y 106.188,Z 584.948,A -85,B 0,C 180,E1 -29513.059,E2 -29513.059} C_VEL
LIN {X 0,Y 106.685,Z 583.938,A -85,B 0,C 180,E1 -29516.223,E2 -29516.223} C_VEL
LIN {X 0,Y 107.342,Z 583.092,A -85,B 0,C 180,E1 -29520,E2 -29520} C_VEL
LIN {X 0,Y 107.083,Z 583.63,A -85,B 0,C 180,E1 -29523.763,E2 -29523.763} C_VEL
LIN {X 0,Y 106.605,Z 585.135,A -85,B 0,C 180,E1 -29528.587,E2 -29528.587} C_VEL
LIN {X 0,Y 106.414,Z 586.278,A -85,B 0,C 180,E1 -29531.427,E2 -29531.427} C_VEL
LIN {X 0,Y 105.759,Z 588.554,A -85,B 0,C 180,E1 -29535.415,E2 -29535.415} C_VEL
LIN {X 0,Y 104.051,Z 590.472,A -85,B 0,C 180,E1 -29536.295,E2 -29536.295} C_VEL
LIN {X 0,Y 94.641,Z 598.92,A -85,B 0,C 180,E1 -29538.79,E2 -29538.79} C_VEL
LIN {X 0,Y 85.231,Z 606.142,A -85,B 0,C 180,E1 -29541.946,E2 -29541.946} C_VEL
LIN {X 0,Y 74.67,Z 613.04,A -85,B 0,C 180,E1 -29546.617,E2 -29546.617} C_VEL
LIN {X 0,Y 64.739,Z 618.549,A -85,B 0,C 180,E1 -29552.874,E2 -29552.874} C_VEL
LIN {X 0,Y 55.992,Z 622.726,A -85,B 0,C 180,E1 -29561.154,E2 -29561.154} C_VEL
LIN {X 0,Y 47.704,Z 626.144,A -85,B 0,C 180,E1 -29573.906,E2 -29573.906} C_VEL
LIN {X 0,Y 42.575,Z 628.164,A -85,B 0,C 180,E1 -29590.735,E2 -29590.735} C_VEL
LIN {X 0,Y 41.208,Z 628.826,A -85,B 0,C 180,E1 -29610.012,E2 -29610.012} C_VEL
LIN {X 0,Y 42.58,Z 628.127,A -85,B 0,C 180,E1 -29629.288,E2 -29629.288} C_VEL
LIN {X 0,Y 47.713,Z 626.076,A -85,B 0,C 180,E1 -29646.113,E2 -29646.113} C_VEL
LIN {X 0,Y 56.038,Z 622.629,A -85,B 0,C 180,E1 -29658.819,E2 -29658.819} C_VEL
LIN {X 0,Y 58.261,Z 621.656,A -85,B 0,C 180,E1 -29661.198,E2 -29661.198} C_VEL
LIN {X 0,Y 59.997,Z 620.546,A -85,B 0,C 180,E1 -29664.149,E2 -29664.149} C_VEL
LIN {X 0,Y 54.108,Z 619.108,A -85,B 0,C 180,E1 -29684.944,E2 -29684.944} C_VEL
LIN {X 0,Y 70.055,Z 614.833,A -85,B 0,C 180,E1 -29728.46,E2 -29728.46} C_VEL
LIN {X 0,Y 68.628,Z 616.021,A -85,B 0,C 180,E1 -29730.8,E2 -29730.8} C_VEL
LIN {X 0,Y 58.816,Z 620.99,A -85,B 0,C 180,E1 -29739.028,E2 -29739.028} C_VEL
LIN {X 0,Y 51.898,Z 623.933,A -85,B 0,C 180,E1 -29747.37,E2 -29747.37} C_VEL
LIN {X 0,Y 45.012,Z 626.647,A -85,B 0,C 180,E1 -29762.057,E2 -29762.057} C_VEL
LIN {X 0,Y 41.486,Z 628.003,A -85,B 0,C 180,E1 -29780.234,E2 -29780.234} C_VEL
LIN {X 0,Y 41.283,Z 628.179,A -85,B 0,C 180,E1 -29789.988,E2 -29789.988} C_VEL
LIN {X 0,Y 42.761,Z 627.536,A -85,B 0,C 180,E1 -29809.178,E2 -29809.178} C_VEL
LIN {X 0,Y 48.206,Z 625.469,A -85,B 0,C 180,E1 -29826.174,E2 -29826.174} C_VEL
LIN {X 0,Y 56.348,Z 622.158,A -85,B 0,C 180,E1 -29838.433,E2 -29838.433} C_VEL
LIN {X 0,Y 66.534,Z 617.275,A -85,B 0,C 180,E1 -29847.661,E2 -29847.661} C_VEL
LIN {X 0,Y 67.662,Z 616.68,A -85,B 0,C 180,E1 -29848.466,E2 -29848.466} C_VEL
LIN {X 0,Y 71.541,Z 614.414,A -85,B 0,C 180,E1 -29851.642,E2 -29851.642} C_VEL
LIN {X 0,Y 77.18,Z 610.417,A -85,B 0,C 180,E1 -29857.149,E2 -29857.149} C_VEL
LIN {X 0,Y 83.181,Z 605.836,A -85,B 0,C 180,E1 -29861.735,E2 -29861.735} C_VEL
LIN {X 0,Y 87.402,Z 602.661,A -85,B 0,C 180,E1 -29863.498,E2 -29863.498} C_VEL
LIN {X 0,Y 97.565,Z 594.533,A -85,B 0,C 180,E1 -29866.14,E2 -29866.14} C_VEL
LIN {X 0,Y 99.288,Z 592.624,A -85,B 0,C 180,E1 -29867.739,E2 -29867.739} C_VEL
LIN {X 0,Y 99.986,Z 591.505,A -85,B 0,C 180,E1 -29869.723,E2 -29869.723} C_VEL
LIN {X 0,Y 100.523,Z 590.49,A -85,B 0,C 180,E1 -29871.962,E2 -29871.962} C_VEL
LIN {X 0,Y 101.443,Z 589.012,A -85,B 0,C 180,E1 -29876.027,E2 -29876.027} C_VEL
LIN {X 0,Y 102.214,Z 588.128,A -85,B 0,C 180,E1 -29880,E2 -29880} C_VEL
LIN {X 0,Y 101.898,Z 588.688,A -85,B 0,C 180,E1 -29883.955,E2 -29883.955} C_VEL
LIN {X 0,Y 101.437,Z 589.832,A -85,B 0,C 180,E1 -29887.965,E2 -29887.965} C_VEL
LIN {X 0,Y 100.802,Z 591.775,A -85,B 0,C 180,E1 -29892.579,E2 -29892.579} C_VEL
LIN {X 0,Y 97.557,Z 594.728,A -85,B 0,C 180,E1 -29893.484,E2 -29893.484} C_VEL
LIN {X 0,Y 87.664,Z 602.646,A -85,B 0,C 180,E1 -29895.86,E2 -29895.86} C_VEL
LIN {X 0,Y 78.04,Z 609.229,A -85,B 0,C 180,E1 -29899.008,E2 -29899.008} C_VEL
LIN {X 0,Y 68.675,Z 614.687,A -85,B 0,C 180,E1 -29902.944,E2 -29902.944} C_VEL
LIN {X 0,Y 56.968,Z 620.407,A -85,B 0,C 180,E1 -29910.299,E2 -29910.299} C_VEL
LIN {X 0,Y 46.587,Z 624.56,A -85,B 0,C 180,E1 -29921.054,E2 -29921.054} C_VEL
LIN {X 0,Y 38.559,Z 627.269,A -85,B 0,C 180,E1 -29936.869,E2 -29936.869} C_VEL
LIN {X 0,Y 34.404,Z 628.609,A -85,B 0,C 180,E1 -29958.228,E2 -29958.228} C_VEL
LIN {X 0,Y 34.101,Z 628.771,A -85,B 0,C 180,E1 -29970.015,E2 -29970.015} C_VEL
LIN {X 0,Y 35.941,Z 628.071,A -85,B 0,C 180,E1 -29993.038,E2 -29993.038} C_VEL
LIN {X 0,Y 42.153,Z 626.019,A -85,B 0,C 180,E1 -30011.845,E2 -30011.845} C_VEL
LIN {X 0,Y 51.616,Z 622.572,A -85,B 0,C 180,E1 -30024.798,E2 -30024.798} C_VEL
LIN {X 0,Y 51.328,Z 622.328,A -85,B 0,C 180,E1 -30026.792,E2 -30026.792} C_VEL
LIN {X 0,Y 47.32,Z 620.968,A -85,B 0,C 180,E1 -30051.46,E2 -30051.46} C_VEL
LIN {X 0,Y 60.764,Z 618.136,A -85,B 0,C 180,E1 -30087.559,E2 -30087.559} C_VEL
LIN {X 0,Y 57.316,Z 619.837,A -85,B 0,C 180,E1 -30090.854,E2 -30090.854} C_VEL
LIN {X 0,Y 51.95,Z 622.099,A -85,B 0,C 180,E1 -30095.721,E2 -30095.721} C_VEL
LIN {X 0,Y 42.486,Z 625.52,A -85,B 0,C 180,E1 -30108.557,E2 -30108.557} C_VEL
LIN {X 0,Y 36.118,Z 627.549,A -85,B 0,C 180,E1 -30127.082,E2 -30127.082} C_VEL
LIN {X 0,Y 34.173,Z 628.235,A -85,B 0,C 180,E1 -30149.985,E2 -30149.985} C_VEL
LIN {X 0,Y 36.106,Z 627.592,A -85,B 0,C 180,E1 -30172.895,E2 -30172.895} C_VEL
LIN {X 0,Y 42.446,Z 625.6,A -85,B 0,C 180,E1 -30191.459,E2 -30191.459} C_VEL
LIN {X 0,Y 51.898,Z 622.213,A -85,B 0,C 180,E1 -30204.325,E2 -30204.325} C_VEL
LIN {X 0,Y 63.507,Z 617.085,A -85,B 0,C 180,E1 -30213.471,E2 -30213.471} C_VEL
LIN {X 0,Y 75.113,Z 610.802,A -85,B 0,C 180,E1 -30219.313,E2 -30219.313} C_VEL
LIN {X 0,Y 86.262,Z 603.511,A -85,B 0,C 180,E1 -30223.175,E2 -30223.175} C_VEL
LIN {X 0,Y 87.402,Z 602.661,A -85,B 0,C 180,E1 -30223.498,E2 -30223.498} C_VEL
LIN {X 0,Y 89.653,Z 600.874,A -85,B 0,C 180,E1 -30224.541,E2 -30224.541} C_VEL
LIN {X 0,Y 91.976,Z 598.632,A -85,B 0,C 180,E1 -30226.704,E2 -30226.704} C_VEL
LIN {X 0,Y 93.761,Z 596.567,A -85,B 0,C 180,E1 -30229.72,E2 -30229.72} C_VEL
LIN {X 0,Y 95.015,Z 594.969,A -85,B 0,C 180,E1 -30233,E2 -30233} C_VEL
LIN {X 0,Y 95.517,Z 594.314,A -85,B 0,C 180,E1 -30234.668,E2 -30234.668} C_VEL
LIN {X 0,Y 96.819,Z 592.938,A -85,B 0,C 180,E1 -30240,E2 -30240} C_VEL
LIN {X 0,Y 96.453,Z 593.508,A -85,B 0,C 180,E1 -30244.178,E2 -30244.178} C_VEL
LIN {X 0,Y 95.83,Z 594.731,A -85,B 0,C 180,E1 -30248.434,E2 -30248.434} C_VEL
LIN {X 0,Y 94.245,Z 596.293,A -85,B 0,C 180,E1 -30249.686,E2 -30249.686} C_VEL
